// TwinCAT 3 PLC project Plc
// ProgramVersion: 3.1.4026.21
// libraries:
//   [IIN_Base], * (IIN Solutions Oy)
//   Meca500 Functions, * (Iin Solutions Oy)
//   Tc2_DataExchange, * (Beckhoff Automation GmbH)
//   Tc2_MC2, * (Beckhoff Automation GmbH)
//   Tc2_Standard, * (Beckhoff Automation GmbH)
//   Tc2_System, * (Beckhoff Automation GmbH)
//   Tc2_Utilities, * (Beckhoff Automation GmbH)
//   Tc3_EventLogger, * (Beckhoff Automation GmbH)
//   Tc3_Vision, * (Beckhoff Automation GmbH)
// project tree:
//   DUTs/Com/ ST_MecaHmi.TcDUT, ST_ModuleHmi.TcDUT, ST_Module_PlcCom.TcDUT, ST_Module_PlcComIn.TcDUT, ST_Module_PlcComOut.TcDUT, ST_StationHmi.TcDUT
//   DUTs/ E_MecaStatus.TcDUT, ST_Recipes.TcDUT, ST_Recipe_AssemblyData.TcDUT
//   GVLs/ Color.TcGVL, Err.TcGVL, Trig.TcGVL
//   / PlcTask.TcTTO, PlcTaskVis.TcTTO
//   POUs/ FB_ASMT60Functions.TcPOU, FB_GlueState.TcPOU, MAIN.TcPOU
//   POUs/HP/CURING_STATION/ E_CURING_STATION_SEQUENCE_STEPS.TcDUT, E_CURING_STATION_OPERATION_STATE.TcDUT, FB_CuringStation.TcPOU, ST_CURING_STATION_HMI.TcDUT, ST_CURING_STATION_SERVICE.TcDUT, ST_CURING_STATION_STATE.TcDUT, ST_CURING_STATION_SETTINGS.TcDUT
//   POUs/HP/CURING_STATION/HEATER/ E_CURING_STATION_HEATER_CONTROL_STEPS.TcDUT (not stored), FB_CuringStationHeaterControl.TcPOU, ST_CURING_STATION_HEATER_CONTROL_HMI.TcDUT, ST_CURING_STATION_HEATER_CONTROL_SERVICE.TcDUT, ST_CURING_STATION_HEATER_CONTROL_STATE.TcDUT, ST_CURING_STATION_HEATER_CONTROL_STATIC_SETTINGS.TcDUT
//   POUs/HP/CURING_STATION/VISION/Coupler/ E_COUPLER_PROCESSOR_STEPS.TcDUT, FB_CouplerImageProcessor.TcPOU, I_ImageProcessor.TcIO, ST_COUPLER_DETECT_SETTINGS.TcDUT
//   POUs/HP/CURING_STATION/VISION/ E_GIGE_CAM_HANDLER_SEQ_STEPS.TcDUT, E_NORMAL_CAM_HANDLER_SEQ_STEPS.TcDUT, FB_GigECamHandler.TcPOU, FB_CuringStationCameraHandler.TcPOU, ST_LASER_TEST_SETTINGS.TcDUT, ST_NORMAL_CAM_HANDLER_HMI.TcDUT, ST_NORMAL_CAM_HANDLER_SERVICE.TcDUT, ST_NORMAL_CAM_HANDLER_SETTINGS.TcDUT, ST_TEST_SETTING.TcDUT, ST_UNDERLIGHT_TEST_SETTINGS.TcDUT, VISION_PARAMS.TcGVL
//   POUs/HP/CURING_STATION/VISION/GenericCameraHandler/ E_GENERIC_CAM_HANDLER_SEQ_STEPS.TcDUT, FB_GenericCameraHandler.TcPOU
//   POUs/HP/CURING_STATION/VISION/HelperFunctions/ FC_CalculateCenterPoint.TcPOU, FC_CalculateYCenterPoint.TcPOU (not stored), FC_ExtractFromContainerAndCalculateAvg.TcPOU
//   POUs/HP/CURING_STATION/VISION/Mirror/ E_MIRROR_PROCESSOR_STEPS.TcDUT, FB_MirrorImageProcessor.TcPOU, FC_GetCameraScalingFactor.TcPOU, I_MirrorImageProcessor.TcIO, ST_MIRROR_DETECT_SETTINGS.TcDUT
//   POUs/HP/GVL/ HEATER_CONTROL_SETTINGS.TcGVL, HMI.TcGVL, MAIN_VISION_COMM_VARS.TcGVL
//   POUs/HP/ P_Heaters.TcPOU
//   POUs/Meca500/ FB_linearAxisFunctions.TcPOU, FB_MecaStateMachine.TcPOU
//   POUs/Meca500/Op/ E_CurrentState.TcDUT, E_OperatingState.TcDUT, FB_GluingTipPositioning.TcPOU, FB_ManualControl.TcPOU, FB_MecaConf.TcPOU, FB_Operating.TcPOU
//   POUs/Meca500/Op/PoseData/ ST_GluetipCoordinates.TcDUT, ST_GluingPoses.TcDUT, ST_Sts_PoseData.TcDUT, ST_Sts1_PoseData.TcDUT, ST_Sts10_PoseData.TcDUT, ST_Sts2_PoseData.TcDUT, ST_Sts3_PoseData.TcDUT, ST_Sts4_PoseData.TcDUT, ST_Sts5_PoseData.TcDUT, ST_Sts6_PoseData.TcDUT, ST_Sts7_PoseData.TcDUT, ST_Sts8_PoseData.TcDUT, ST_Sts9_PoseData.TcDUT
//   POUs/Meca500/Op/PoseData/Type/ AL82027.TcDUT, AL86068.TcDUT, AL200663.TcDUT, AL200665.TcDUT, AL200664.TcDUT, AL200662.TcDUT
//   POUs/Sts/Com/ FB_DataExchangeRead.TcPOU, FB_RecipeDataExchange.TcPOU, ST_Stations.TcDUT, ST_Sts_PlcCom.TcDUT, ST_Sts_PlcComIn.TcDUT, ST_Sts_PlcComOut.TcDUT
//   POUs/Sts/Datalog/ FB_Datalogger2.TcPOU, FB_Datalogger3.TcPOU, FB_EventLogger.TcPOU, ST_LogEntry.TcDUT
//   POUs/Sts/DUT/ E_MovementState.TcDUT, E_StepperState.TcDUT, E_StsActState.TcDUT, ST_AngleData.TcDUT, ST_Sts_DetectionData.TcDUT, ST_Vis_Laser.TcDUT, ST_Vis_Mirror.TcDUT
//   POUs/Sts/ FB_HeaterControl.TcPOU, FB_Stepper.TcPOU, FB_StsAct.TcPOU
//   POUs/Sts/Vis/ FB_PosImgSts.TcPOU
//   POUs/VisMain/ FB_MidStaion.TcPOU, FB_InfeedCam.TcPOU, FB_OutfeedCam.TcPOU, FB_RejectCam.TcPOU, MAIN_VISION.TcPOU, ST_CouplerImagingData.TcDUT, ST_PalletImagingData.TcDUT

CONFIGURATION Plc
    RESOURCE PLC ON TwinCAT3
        TASK PlcTask(INTERVAL := T#10ms, PRIORITY := 20);
        TASK PlcTaskVis(INTERVAL := T#150ms, PRIORITY := 1);
        PROGRAM MAIN WITH PlcTask : MAIN;
        PROGRAM MAIN_VISION WITH PlcTaskVis : MAIN_VISION;
    END_RESOURCE
END_CONFIGURATION

// ---- DUTs/Com/ST_MecaHmi.TcDUT
TYPE ST_MecaHmi :
STRUCT
	
	bJogToPose			: BOOL;
	aPoseDirect			: ARRAY [1..6] OF REAL;
	bHomeAxis			: BOOL;
	bSetGripperWidth	: BOOL;
	rGripperWidth		: REAL;

// Direct control buttons to robot
	bActivate			: BOOL;
	bDeactivate			: BOOL;
	bErrorReset			: BOOL;
	bManualJog			: BOOL;
	bClearMove			: BOOL;
	bPauseMotion		: BOOL;
	bResumeMotion		: BOOL;
	bDisableEtherCat	: BOOL;
	bToggleGripper		: BOOL;
	bRecoveryMode		: BOOL;

	bJogXPositive		: BOOL;
	bJogXNegative		: BOOL;
	bJogYPositive		: BOOL;
	bJogYNegative		: BOOL;
	bJogZPositive		: BOOL;
	bJogZNegative		: BOOL;
	bJogRxPositive		: BOOL;
	bJogRxNegative		: BOOL;
	bJogRyPositive		: BOOL;
	bJogRyNegative		: BOOL;
	bJogRzPositive		: BOOL;
	bJogRzNegative		: BOOL;
	rJogSpeed			: REAL := 10;
	aCurrentPose		: ARRAY [1..6] OF REAL;
	bJogLinearPositive	: BOOL;
	bJogLinearNegative	: BOOL;
	bLinearJogScreenActive	: BOOL;
	bManualAbsMove : BOOL;
	rManualTargetPos	: REAL;
	
END_STRUCT
END_TYPE

// ---- DUTs/Com/ST_ModuleHmi.TcDUT
TYPE ST_ModuleHmi :
STRUCT
	
	MecaHmi 					: ST_MecaHmi;
	Stations					: ST_StationHmi;
	bModuleProductionStart		: BOOL; // Is always active if assemblies are active
	bModulePlayPause 			: BOOL; // Only used for glue remove
	bProductionStart1To5 		: BOOL; // 
	bProductionStart6To10		: BOOL;
	bProductionStageCompleted	: BOOL; // To indicate that assemblies of 1 to 5 or 6 to 10 are set and more assemblies can be inserted
	bModuleProductionStop		: BOOL;
	bModuleStartup				: BOOL;
	bModuleStartupDone			: BOOL;
	bModuleFault				: BOOL;
	bResetCommunication			: BOOL;
	bResetModuleFault			: BOOL;
	bPowerOff					: BOOL;
	bClearAlarms				: BOOL;
	sOperatingStatus			: STRING;
	bProductionStartFailure		: BOOL;
	bOpenAllLocks				: BOOL;
	bAcOk						: BOOL;
	
	bGlueDispensing				: BOOL;
	bToggleDispensingPressure	: BOOL;
	bDispensingPressed			: BOOL;
	bStartDetection				: BOOL;
	bAllowManDispensing			: BOOL;
	bDetectionSucceeded			: BOOL;
	sTimeSinceDispensing		: STRING;
	bDispensingStageDone		: BOOL;
	
END_STRUCT
END_TYPE

// ---- DUTs/Com/ST_Module_PlcCom.TcDUT
TYPE ST_Module_PlcCom :
STRUCT
	
	stPlcComIn		AT %I*: ST_Module_PlcComIn;
	stPlcComOut		AT %Q*: ST_Module_PlcComOut;

END_STRUCT
END_TYPE

// ---- DUTs/Com/ST_Module_PlcComIn.TcDUT
TYPE ST_Module_PlcComIn :
STRUCT
	bEstopOk	: BOOL;
	bSafetyOk  : BOOL;
	bUpsStatusOk	: BOOL;	
	bLinearAxisHomingSensor : BOOL;
	bRobotGripperSensor : BOOL;
	bRobotPower	: BOOL;
	
	bGlueDoorUpperLockOpen		: BOOL;
	bGlueDoorUpperLockClosed	: BOOL;
	bGlueDoorLowerLockOpen		: BOOL;
	bGlueDoorLowerLockClosed	: BOOL;
	
	bMainDoorLockOpen			: BOOL;
	bMainDoorLockClosed			: BOOL;
	bPassLockOpen				: BOOL;
	bPassLockClosed				: BOOL;
	bInfeedLockOpen				: BOOL;
	bInfeedLockClosed			: BOOL;
	bRejectLockOpen				: BOOL;
	bRejectLockClosed			: BOOL;
	
	bUpsAlarm					: BOOL;
	bAcOk						: BOOL;
	iModuleTemp					: INT;
	bGlueStopHome				: BOOL;
END_STRUCT
END_TYPE

// ---- DUTs/Com/ST_Module_PlcComOut.TcDUT
TYPE ST_Module_PlcComOut :
STRUCT
	bTriggerGluing1			: BOOL;
	bLaserPointers1To5		: BOOL;
	bLaserPointers5To10		: BOOL;
	bResetButtonLight		: BOOL;
	bMecaReset				: BOOL;
	bRobotSwStop			: BOOL;
	
	bRingLightGlue			: BOOL;
	bRingLightInfeed		: BOOL;
	bRingLightPass			: BOOL;
	bRingLightReject		: BOOL;
	
	bGlueDoorLock			: BOOL;
	bHatchesLock			: BOOL;
	bPowerOff				: BOOL;
	bGlueStopValve			: BOOL;
	bGlueSelectingValve		: BOOL;
END_STRUCT
END_TYPE

// ---- DUTs/Com/ST_StationHmi.TcDUT
TYPE ST_StationHmi :
STRUCT
		
	bActivateStation1 : BOOL := TRUE;
	bActivateStation2 : BOOL := TRUE;
	bActivateStation3 : BOOL := TRUE;
	bActivateStation4 : BOOL := TRUE;
	bActivateStation5 : BOOL := TRUE;
	bActivateStation6 : BOOL := TRUE;
	bActivateStation7 : BOOL := TRUE;
	bActivateStation8 : BOOL := TRUE;
	bActivateStation9 : BOOL := TRUE;
	bActivateStation10 : BOOL := TRUE;
	
	tAssemmblyTime1				: STRING;
	tAssemmblyTime2				: STRING;
	tAssemmblyTime3				: STRING;
	tAssemmblyTime4				: STRING;
	tAssemmblyTime5				: STRING;
	tAssemmblyTime6				: STRING;
	tAssemmblyTime7				: STRING;
	tAssemmblyTime8				: STRING;
	tAssemmblyTime9				: STRING;
	tAssemmblyTime10			: STRING;
	
	bReleaseHolders1			: BOOL;
	bReleaseHolders2			: BOOL;
	bReleaseHolders3			: BOOL;
	bReleaseHolders4			: BOOL;
	bReleaseHolders5			: BOOL;
	bReleaseHolders6			: BOOL;
	bReleaseHolders7			: BOOL;
	bReleaseHolders8			: BOOL;
	bReleaseHolders9			: BOOL;
	bReleaseHolders10			: BOOL;
	
END_STRUCT
END_TYPE

// ---- DUTs/E_MecaStatus.TcDUT
{attribute 'qualified_only'}
{attribute 'strict'}
{attribute 'to_string'}
TYPE E_MecaStatus :
(
	Offline,
	Conf,
	Idle,
	Operating,
	Home,
	HmiManual,
	GluingpPos
);
END_TYPE

// ---- DUTs/ST_Recipes.TcDUT
TYPE ST_Recipes :
STRUCT
	Station1To5		: ST_Recipe_AssemblyData;
	Station5To10	: ST_Recipe_AssemblyData;
END_STRUCT
END_TYPE

// ---- DUTs/ST_Recipe_AssemblyData.TcDUT
TYPE ST_Recipe_AssemblyData :
STRUCT
	rGalvoThickness			: REAL;
	rMirrorDimensions : ARRAY [0..3] OF REAL; //[0] Width at mirror girp center position (gripperWidth), [1] Width, [2] height, [3] Thickness
 	
	// To enable new mirror variations to be added only based on offset values
	rMirrorGripPointOffsetToEdgeX	: REAL; // Distance from grip centerpoint to mirror edge on the direction of the gluing side
	rMirrorCenterOffsetToWeightCenterY : REAL; // Distance from mirror weight centerpoint to mirror width centerpoint.
	rLaserPointSetValue	: REAL;
	rCouplerGroveDepth	: REAL; // Depth from CAD files of the couplers
	// Coupler detection variables
	rThreshold			: LREAL;
	aStartPointCoupler					: TcVnPoint2_REAL;
	aEndPointCoupler					: TcVnPoint2_REAL;
	rSearchLineDist							: REAL;
	//
	wPalletBinary		: WORD;
	sAssemblyType	: STRING;
	sMotorType	: STRING;
	sMirrorType	: STRING;
	sGlueType	: STRING;
	sCouplerType : STRING;
	
	// for data exchange
	bTrigCam1	: BOOL;
	bTrigCam2	: BOOL;
	bTrigCam3	: BOOL;
	bTrigCam4	: BOOL;
	bTrigCam5	: BOOL;
	bTrigCam6	: BOOL;
	bTrigCam7	: BOOL;
	bTrigCam8	: BOOL;
	bTrigCam9	: BOOL;
	bTrigCam10	: BOOL;
	
END_STRUCT
END_TYPE

// ---- POUs/HP/CURING_STATION/E_CURING_STATION_SEQUENCE_STEPS.TcDUT
{attribute 'qualified_only'}
{attribute 'strict'}
{attribute 'to_string'}
TYPE E_CURING_STATION_SEQUENCE_STEPS :
(
	INIT := 0,
	
	STARTUP_TEST_DO_ECCENTRIC_WHEEL_HOMING,
	
	STARTUP_TEST_TEST_SLIDER_TO_WORK,
	STARTUP_TEST_TEST_SLIDER_TO_HOME,
	
	STARTUP_TEST_TEST_GRIPPER_TO_WORK,
	STARTUP_TEST_TEST_GRIPPER_TO_HOME,
	
	STARTUP_TEST_TEST_UNDERLIGHT,
	
	STARTUP_TEST_TEST_LASER,
	
	STARTUP_TEST_TEST_HEATER,

	STARTUP_TEST_DONE,

	STARTUP_TEST_FAIL,	
	
	OPERATIONAL
	
);
END_TYPE

// ---- POUs/HP/CURING_STATION/E_CURING_STATION_OPERATION_STATE.TcDUT
{attribute 'qualified_only'}
{attribute 'strict'}
{attribute 'to_string'}
TYPE E_CURING_STATION_OPERATION_STATE :
(
	INACTIVE := 0,
	
	OPERATIONAL,
	
	FAULTED
);
END_TYPE

// ---- POUs/HP/CURING_STATION/HEATER/ST_CURING_STATION_HEATER_CONTROL_HMI.TcDUT
TYPE ST_CURING_STATION_HEATER_CONTROL_HMI :
STRUCT
	state:				ST_CURING_STATION_HEATER_CONTROL_STATE;
	service:			ST_CURING_STATION_HEATER_CONTROL_SERVICE;
	
	ai:						ST_AI_HMI;
//	regularThermostat:		ST_THERMOSTAT_HMI;
	specialThermostat:		ST_TIME_PROPORTIONAL_THERMOSTAT_HMI;
END_STRUCT
END_TYPE

// ---- POUs/HP/CURING_STATION/HEATER/ST_CURING_STATION_HEATER_CONTROL_SERVICE.TcDUT
TYPE ST_CURING_STATION_HEATER_CONTROL_SERVICE :
STRUCT
	
END_STRUCT
END_TYPE

// ---- POUs/HP/CURING_STATION/HEATER/ST_CURING_STATION_HEATER_CONTROL_STATE.TcDUT
TYPE ST_CURING_STATION_HEATER_CONTROL_STATE :
STRUCT
	enabled:					BOOL;
	heat:						BOOL;
	fan:						BOOL;
	tempInC:					REAL;
//		tempInF:					REAL;
	testTemperatureReached:		BOOL; 
	workTemperatureReached:		BOOL;
	stationId:					UDINT; 
END_STRUCT
END_TYPE

// ---- POUs/HP/CURING_STATION/HEATER/ST_CURING_STATION_HEATER_CONTROL_STATIC_SETTINGS.TcDUT
TYPE ST_CURING_STATION_HEATER_CONTROL_STATIC_SETTINGS :
STRUCT
	testTemperature:			REAL := 28.0;
	workTemperature:			REAL := 50.0;
	hysteresis:					REAL := 2.0;	// If temp within this value, temp is 'reached'
	
	pFactor:					REAL := 3;		// Temp diff * pFactor = power output (just like a PID controller but without the ID)
	minPowerProcent:			REAL := 20;		// If this were a PID controller, we need 20% to keep the constant heat (at target setpoint)
	maxPowerProcent:			REAL := 80;		// To limit the output (in case the heating element is too powerfull)

	cycleTime:					TIME := T#20S;	// 100% control = HEAT is on for this amount of cycle time, 50% results in 10sec ON and 10s OFF
	nrOfStations:				UDINT := 10;	// Used to calculate a start delay for the heaters to go on -> so FUSE won't blow
END_STRUCT
END_TYPE

// ---- POUs/HP/CURING_STATION/ST_CURING_STATION_HMI.TcDUT
TYPE ST_CURING_STATION_HMI :
STRUCT
	state:			ST_CURING_STATION_STATE;
	service:		ST_CURING_STATION_SERVICE;
	settings:		ST_CURING_STATION_SETTINGS;
	
	cyls:			ARRAY[0..1] OF ST_CYL_HMI;
	heater:			ST_CURING_STATION_HEATER_CONTROL_HMI;
END_STRUCT
END_TYPE

// ---- POUs/HP/CURING_STATION/ST_CURING_STATION_SERVICE.TcDUT
TYPE ST_CURING_STATION_SERVICE :
STRUCT
	enable:	BOOL;		// Setting on/off will enable the station
END_STRUCT
END_TYPE

// ---- POUs/HP/CURING_STATION/ST_CURING_STATION_STATE.TcDUT
TYPE ST_CURING_STATION_STATE :
STRUCT
	stationId:				UDINT; 
	operationState:			E_CURING_STATION_OPERATION_STATE;
END_STRUCT
END_TYPE

// ---- POUs/HP/CURING_STATION/ST_CURING_STATION_SETTINGS.TcDUT
TYPE ST_CURING_STATION_SETTINGS :
STRUCT
END_STRUCT
END_TYPE

// ---- POUs/HP/CURING_STATION/VISION/Coupler/E_COUPLER_PROCESSOR_STEPS.TcDUT
{attribute 'qualified_only'}
{attribute 'strict'}
{attribute 'to_string'}
TYPE E_COUPLER_PROCESSOR_STEPS :
(
	INIT := 0,
	
	LOCATE_EDGE1,
	
	LOCATE_EDGE2,

	LOCATE_EDGE3,
	
	DRAW_POINTS,
	
	MAKE_DISPLAYABLE,
	
	DONE,
	
	ERROR,
	
	END
	
);
END_TYPE

// ---- POUs/HP/CURING_STATION/VISION/Coupler/ST_COUPLER_DETECT_SETTINGS.TcDUT
TYPE ST_COUPLER_DETECT_SETTINGS :
STRUCT
//	startPoint:		TcVnPoint2_REAL := [1000, 550];
//	endPoint:		TcVnPoint2_REAL := [550, 1000];
	
//	minStrength:	REAL := 45;
//	searchLines:	UDINT := 5;
END_STRUCT
END_TYPE

// ---- POUs/HP/CURING_STATION/VISION/E_GIGE_CAM_HANDLER_SEQ_STEPS.TcDUT
{attribute 'qualified_only'}
{attribute 'strict'}
{attribute 'to_string'}
TYPE E_GIGE_CAM_HANDLER_SEQ_STEPS :
(
	INIT,
	
	RESET_CAMERA,
	
	READY_FOR_OPERATION,
	
	TRIGGER_CAMERA,
	
	START_ACQUISITION,
	
	ACQUIRING,
	
	DO_COLOR_CONVERSION,
	
	ACQUIRED,
	
	ERROR,
	
	DONE,
	
	END
);
END_TYPE

// ---- POUs/HP/CURING_STATION/VISION/E_NORMAL_CAM_HANDLER_SEQ_STEPS.TcDUT
{attribute 'qualified_only'}
{attribute 'strict'}
{attribute 'to_string'}
TYPE E_NORMAL_CAM_HANDLER_SEQ_STEPS :
(
	INIT := 0,

	UNDER_LIGHT_TEST_ENABLE_LIGHT,
	UNDER_LIGHT_TEST_IMAGE_ACQUIRE,
	UNDER_LIGHT_TEST_IMAGE_PROCESSING,
	UNDER_LIGHT_TEST_OK,
	UNDER_LIGHT_TEST_FAILED,

	LASER_LIGHT_TEST_ENABLE_LIGHT,
	LASER_LIGHT_TEST_IMAGE_ACQUIRE,
	LASER_LIGHT_TEST_IMAGE_PROCESSING,
	LASER_LIGHT_TEST_OK,
	LASER_LIGHT_TEST_FAILED,
	
	COUPLER_DETECT_ENABLE_LIGHT,
	COUPLER_DETECT_IMAGE_ACQUIRE,
	COUPLER_DETECT_IMAGE_PROCESSING,
	COUPLER_DETECT_DONE,
	COUPLER_DETECT_FAILED,

	MIRROR_DETECT_ENABLE_LIGHT,
	MIRROR_DETECT_IMAGE_ACQUIRE,
	MIRROR_DETECT_IMAGE_PROCESSING,
	MIRROR_DETECT_DONE,
	MIRROR_DETECT_FAILED,
	
	
	END
);
END_TYPE

// ---- POUs/HP/CURING_STATION/VISION/GenericCameraHandler/E_GENERIC_CAM_HANDLER_SEQ_STEPS.TcDUT
{attribute 'qualified_only'}
{attribute 'strict'}
{attribute 'to_string'}
TYPE E_GENERIC_CAM_HANDLER_SEQ_STEPS :
(
	INIT := 0,

	UNDER_LIGHT_TEST_ENABLE_LIGHT,
	UNDER_LIGHT_TEST_IMAGE_ACQUIRE,
	UNDER_LIGHT_TEST_IMAGE_PROCESSING,
	UNDER_LIGHT_TEST_OK,
	UNDER_LIGHT_TEST_FAILED,

	LASER_LIGHT_TEST_ENABLE_LIGHT,
	LASER_LIGHT_TEST_IMAGE_ACQUIRE,
	LASER_LIGHT_TEST_IMAGE_PROCESSING,
	LASER_LIGHT_TEST_OK,
	LASER_LIGHT_TEST_FAILED,
	
	COUPLER_DETECT_ENABLE_LIGHT,
	COUPLER_DETECT_IMAGE_ACQUIRE,
	COUPLER_DETECT_IMAGE_PROCESSING,
	COUPLER_DETECT_DONE,
	COUPLER_DETECT_FAILED,

	MIRROR_DETECT_ENABLE_LIGHT,
	MIRROR_DETECT_IMAGE_ACQUIRE,
	MIRROR_DETECT_IMAGE_PROCESSING,
	MIRROR_DETECT_DONE,
	MIRROR_DETECT_FAILED,
	
	
	END
);
END_TYPE

// ---- POUs/HP/CURING_STATION/VISION/Mirror/E_MIRROR_PROCESSOR_STEPS.TcDUT
{attribute 'qualified_only'}
{attribute 'strict'}
{attribute 'to_string'}
TYPE E_MIRROR_PROCESSOR_STEPS :
(
	INIT := 0,
	
	CALC_CENTER_POINT_OFFSET,
	
	FIND_UPPER_EDGE,
	
	FIND_LOWER_EDGE,

	DRAW_POINTS,
	
	MAKE_DISPLAYABLE,
	
	DONE,
	
	ERROR,
	
	END
	
);
END_TYPE

// ---- POUs/HP/CURING_STATION/VISION/Mirror/ST_MIRROR_DETECT_SETTINGS.TcDUT
TYPE ST_MIRROR_DETECT_SETTINGS :
STRUCT
//	startPoint:		TcVnPoint2_REAL := [1000, 550];
//	endPoint:		TcVnPoint2_REAL := [550, 1000];
	
//	minStrength:	REAL := 45;
//	searchLines:	UDINT := 5;
END_STRUCT
END_TYPE

// ---- POUs/HP/CURING_STATION/VISION/ST_LASER_TEST_SETTINGS.TcDUT
TYPE ST_LASER_TEST_SETTINGS :
STRUCT
	height:		UDINT := 20;
	width:		UDINT := 20;
	x:			UDINT := 800;
	y:			UDINT := 900;
	
	threshold:	LREAL := 230;		// Average pixel value for the test to be successfull
END_STRUCT
END_TYPE

// ---- POUs/HP/CURING_STATION/VISION/ST_NORMAL_CAM_HANDLER_HMI.TcDUT
TYPE ST_NORMAL_CAM_HANDLER_HMI :
STRUCT
END_STRUCT
END_TYPE

// ---- POUs/HP/CURING_STATION/VISION/ST_NORMAL_CAM_HANDLER_SERVICE.TcDUT
TYPE ST_NORMAL_CAM_HANDLER_SERVICE :
STRUCT
	doUnderLightTest:		BOOL;
	doLaserTest:			BOOL;
END_STRUCT
END_TYPE

// ---- POUs/HP/CURING_STATION/VISION/ST_NORMAL_CAM_HANDLER_SETTINGS.TcDUT
TYPE ST_NORMAL_CAM_HANDLER_SETTINGS :
STRUCT
	underLightTest:	ST_UNDERLIGHT_TEST_SETTINGS;
	laserTest:		ST_LASER_TEST_SETTINGS;
END_STRUCT
END_TYPE

// ---- POUs/HP/CURING_STATION/VISION/ST_TEST_SETTING.TcDUT
TYPE ST_TEST_SETTING :
STRUCT
	height:		UDINT;
	width:		UDINT;
	x:			UDINT;
	y:			UDINT;
END_STRUCT
END_TYPE

// ---- POUs/HP/CURING_STATION/VISION/ST_UNDERLIGHT_TEST_SETTINGS.TcDUT
TYPE ST_UNDERLIGHT_TEST_SETTINGS :
STRUCT
	height:		UDINT := 200;
	width:		UDINT := 200;
	x:			UDINT := 1800;
	y:			UDINT := 900;
	
	threshold:	LREAL := 230;		// Average pixel value for the test to be successfull
END_STRUCT
END_TYPE

// ---- POUs/Meca500/Op/E_CurrentState.TcDUT
{attribute 'qualified_only'}
{attribute 'strict'}
{attribute 'to_string'}
TYPE E_CurrentState :
(
	Init,
	GalvoHandling,
	MirrorAdj,
	FinishedProduct

);
END_TYPE

// ---- POUs/Meca500/Op/E_OperatingState.TcDUT
{attribute 'qualified_only'}
{attribute 'strict'}
{attribute 'to_string'}
TYPE E_OperatingState :
(
	Init,
	MoveLinAxis,
	SetPoses,
	OperatingGalvo14mm,
	OperatingGalvo10mm,
	MirrorAdjustment,
	FinishedHandling14mm,
	FinishedHandling10mm
);
END_TYPE

// ---- POUs/Meca500/Op/PoseData/ST_GluetipCoordinates.TcDUT
TYPE ST_GluetipCoordinates :
STRUCT
	X : REAL;
	Y : REAL;
	Z : REAL;
END_STRUCT
END_TYPE

// ---- POUs/Meca500/Op/PoseData/ST_GluingPoses.TcDUT
TYPE ST_GluingPoses :
STRUCT
	AL200662: AL200662;
	AL82027: AL82027;
END_STRUCT
END_TYPE

// ---- POUs/Meca500/Op/PoseData/ST_Sts_PoseData.TcDUT
TYPE ST_Sts_PoseData :
STRUCT
	// Pickup positions and pass pallet positions are all station related. So from pallet position 1 it is only possible to place it to curing station 1 and to pass pallet position 1.
	// Positions are claculated with 'Machine cordinate chart' Excel
	
	aPoseSmallMotorPickupSt1 : ARRAY [1..6] OF REAL := [-144.652, 129 , 110.5 , 0, -90 ,0] ; // Pose before gripper in to the pallet picking position
	aPoseSmallMotorPickupSt2 : ARRAY [1..6] OF REAL := [-144.652, 129 , 110.5 , 0, -90 ,0] ; // Pose before gripper grip, or pose after gripper grip
	aPoseSmallMotorPickupSt3 : ARRAY [1..6] OF REAL := [-144.652, 129 , 110.5 , 0, -90 ,0] ; // Pose gripper grip
	
	aPoseSmallMotorPlaceSt1 : ARRAY [1..6] OF REAL; // Pose before Small motor in station
	aPoseSmallMotorPlaceSt2 : ARRAY [1..6] OF REAL; // Pose Small motor in station
	rLinPosPlace : LREAL; // Linear axis position for placing functions for selected station

	aPoseMirrorAdj : ARRAY[1..6] OF REAL; // Pose where final position of left mirror is saved in case position adjustment is needed.
	
	aPoseLargeMotorPickupSt1	: ARRAY [1..6] OF REAL := [-95,-150.45 , 110.5 , 0, -90 ,0]; // POSE BEFORE ACTUAL GRIP POSITION -108.2
	aPoseLargeMotorPickupSt2	: ARRAY [1..6] OF REAL := [-128.2,-150.45 , 110.5 , 0, -90 ,0];// ACTUAL GRIP POSITION
	aPoseLargeMotorPickupSt3	: ARRAY [1..6] OF REAL := [-128.2,-150.45 , 200.5 , 0, -90 ,0];// MOTOR LIFT FROM PALLET
	rLinPosMotorPickup				: LREAL := 120; // Linear axis position for pickup functions for selected station
	
	aPoseLargeMotorPlaceSt1	: ARRAY [1..6] OF REAL := [-144.652, 129 ,165.6645  , -180 , 0 , 90]; // POSE BEFORE ACTULA LEAVING POSITION
	aPoseLargeMotorPlaceSt2	: ARRAY [1..6] OF REAL := [-73.8605, 140 ,165.6645  , -180 , 0 , 90]; // ACTUAL POSITION FOR LEAVING MOTOR AT CURING STATION
	aPoseLargeMotorPlaceSt3	: ARRAY [1..6] OF REAL := [-73.8605, 140 ,200  , -180 , 0 , 90]; // POSE AFTER LEAVING MOTOR AT CURING STATION
	
	aPoseMirrorPickupSt1	: ARRAY [1..6] OF REAL := [-159.1,-91.5 , 200 ,180, 0 ,0]; // POSE BEFORE ACTUAL GRIP POSITION
	aPoseMirrorPickupSt2	: ARRAY [1..6] OF REAL := [-159.1,-91.5 , 186.9757 ,180, 0 ,0];// ACTUAL GRIP POSITION 187.1757
	rLinPosMirrorPickup				: LREAL := 120; // Linear axis position for pickup functions for selected station
	
	aPoseMirrorPlaceSt1	: ARRAY [1..6] OF REAL := [-72, 192.8 ,200.3  , -180 , 0 , 90]; // POSE BEFORE INSERTIN MIRROR IN STATION
	aPoseMirrorPlaceSt2	: ARRAY [1..6] OF REAL := [-72, 192.8 ,173.55  , -180 , 0 , 90]; // POSE MIRROR IN STATION BUT NOT INSERTED TO MOTOR  192.8, 173.45
	aPoseMirrorPlaceSt3	: ARRAY [1..6] OF REAL := [-72, 189.4545 ,173.95  , -180 , 0 , 90]; // POSE MIRROR INSERTED TO MOTOR
 	
// 	aPoseSmallMirrorPlaceSt1	: ARRAY [1..6] OF REAL := [-72, 192.8 ,200.3  , -180 , 0 , 90]; // POSE BEFORE INSERTIN MIRROR IN STATION
// 	aPoseSmallMirrorPlaceSt2	: ARRAY [1..6] OF REAL := [-72, 192.8 ,173.55  , -180 , 0 , 90]; // POSE MIRROR IN STATION BUT NOT INSERTED TO MOTOR  192.8, 173.45
// 	aPoseSmallMirrorPlaceSt3	: ARRAY [1..6] OF REAL := [-72, 189.4545 ,173.95  , -180 , 0 , 90]; // POSE MIRROR INSERTED TO MOTOR
	
	aPosePassedLargeSt1 		: ARRAY [1..6] OF REAL := [-72.2, 189.4545 ,173.95  , -180 , 0 , 90];
	aPosePassedLargeSt2			: ARRAY [1..6] OF REAL := [-72.2, 189.4545 ,173.95  , -180 , 0 , 90];
	aPosePassedLargeSt3			: ARRAY [1..6] OF REAL := [-72.2, 189.4545 ,173.95  , -180 , 0 , 90];
	
	aPosePassedSmallSt1			: ARRAY [1..6] OF REAL := [-72.2, 189.4545 ,173.95  , -180 , 0 , 90];
	aPosePassedSmallSt2			: ARRAY [1..6] OF REAL := [-72.2, 189.4545 ,173.95  , -180 , 0 , 90];
	aPosePassedSmallSt3			: ARRAY [1..6] OF REAL := [-72.2, 189.4545 ,173.95  , -180 , 0 , 90];
	aPosePassedSmallSt4			: ARRAY [1..6] OF REAL := [-72.2, 189.4545 ,173.95  , -180 , 0 , 90];
	
	rLinPosPalletPass : LREAL; // Linear axis position for placing passed assembly for selected station
	rLinPosPalletReject : LREAL; // Linear axis position for placing rejected assembly for selected station
	
END_STRUCT
END_TYPE

// ---- POUs/Meca500/Op/PoseData/ST_Sts1_PoseData.TcDUT
TYPE ST_Sts1_PoseData :
STRUCT
	
	aPoseSmallMotorPickupSt1 : ARRAY [1..6] OF REAL := [-220.552, 67.9 , 150, 180, -20 ,0] ; // Pose before gripper in to the pallet picking position
	aPoseSmallMotorPickupSt2 : ARRAY [1..6] OF REAL := [-220.552, 67.9 , 111.4134, 180, -20 ,0] ;  // Pose before gripper grip, or pose after gripper grip
	aPoseSmallMotorPickupSt3 : ARRAY [1..6] OF REAL := [-222.713, 67.9 , 112.2, 180, -20 ,0] ; //  Pose gripper grip CAN NOT BE MOVEPOSE
	rLinPosSmallMotorPickup				: LREAL := 80; // Linear axis position for pickup functions for selected station
	
	aPoseSmallMotorPlaceSt1 : ARRAY [1..6] OF REAL := [-73.2, 168.6 ,110.6 , 180, 0 ,90] ; // Pose before Small motor in station
	aPoseSmallMotorPlaceSt2 : ARRAY [1..6] OF REAL  := [-73.2, 168.6 ,67.6 , 180, 0 ,90]; // Pose Small motor in station
	rLinPosPlace : LREAL := 10; // Linear axis position for placing functions for selected station

	aPoseMirrorAdj : ARRAY[1..6] OF REAL; // Pose where final position of left mirror is saved in case position adjustment is needed.
	
	aPoseLargeMotorPickupSt1	: ARRAY [1..6] OF REAL := [-124.609, 117.800 , 101.6 , 0, -90 ,0]; // POSE BEFORE ACTUAL GRIP POSITION -108.2
	aPoseLargeMotorPickupSt2	: ARRAY [1..6] OF REAL := [-224.609, 117.800 , 101.6 , 0, -90 ,0];// ACTUAL GRIP POSITION
	aPoseLargeMotorPickupSt3	: ARRAY [1..6] OF REAL := [-224.609, 117.800 , 201.6 , 0, -90 ,0];// MOTOR LIFT FROM PALLET
	rLinPosMotorPickup				: LREAL := 120; // Linear axis position for pickup functions for selected station
	
	aPoseLargeMotorPlaceSt1	: ARRAY [1..6] OF REAL := [-73.3, 80 , 67.6 , 180, 0 ,90]; // POSE BEFORE ACTULA LEAVING POSITION '
	aPoseLargeMotorPlaceSt2	: ARRAY [1..6] OF REAL := [-73.3, 146 , 67.6 , 180, 0 ,90]; // ACTUAL POSITION FOR LEAVING MOTOR AT CURING STATION '
	aPoseLargeMotorPlaceSt3	: ARRAY [1..6] OF REAL := [-73.3, 146 , 100.6 , 180, 0 ,90]; // POSE AFTER LEAVING MOTOR AT CURING STATION '
	
	aPoseMirrorPickupSt1	: ARRAY [1..6] OF REAL := [-158.84, 76.3 , 120, 181, 0 ,0]; // POSE BEFORE ACTUAL GRIP POSITION
	aPoseMirrorPickupSt2	: ARRAY [1..6] OF REAL := [-158.84, 76.3 , 81.55, 181, 0 ,0];// ACTUAL GRIP POSITION 187.1757
	rLinPosMirrorPickup				: LREAL := 80; // Linear axis position for pickup functions for selected station
	
 	aPoseG10MirrorPlaceSt1	: ARRAY [1..6] OF REAL := [-73.3, 190.6 ,117.4 , 180, 0 ,90]; // POSE BEFORE INSERTIN MIRROR IN STATION'
 	aPoseG10MirrorPlaceSt2	: ARRAY [1..6] OF REAL := [-73.3, 188.2 ,70.4 , -180, 0 ,90]; // POSE MIRROR IN STATION BUT NOT INSERTED TO MOTOR '
 	aPoseg10MirrorPlaceSt3	: ARRAY [1..6] OF REAL := [-73.3, 187 ,68.6 , -179, 0 ,90]; // POSE MIRROR INSERTED TO MOTOR'
	
	aPoseG14MirrorPlaceSt1	: ARRAY [1..6] OF REAL := [-73.3, 190.6 ,117.4 , 180, 0 ,90]; // POSE BEFORE INSERTIN MIRROR IN STATION'
	aPoseG14MirrorPlaceSt2	: ARRAY [1..6] OF REAL := [-73.3, 191.6 ,70.4 , -170, 0 ,90]; // POSE MIRROR IN STATION BUT NOT INSERTED TO MOTOR '
	aPoseg14MirrorPlaceSt3	: ARRAY [1..6] OF REAL := [-73.3, 190.1 ,68.6 , -178.5, -0.2 ,90]; // POSE MIRROR INSERTED TO MOTOR'
	
	aPosePassedLargeSt1 		: ARRAY [1..6] OF REAL := [-213.4, 62.25 , 141.45, 180, -20 ,0]; // In and out of pallet
	aPosePassedLargeSt2			: ARRAY [1..6] OF REAL := [-223.4, 62.25 , 101.45, 180, -20 ,0]; // before leaving position
	aPosePassedLargeSt3			: ARRAY [1..6] OF REAL := [-228, 62.25 ,97.79, 180, -20 ,0]; // Leaving position
	
	aPosePassedSmallSt1			: ARRAY [1..6] OF REAL := [-243.3, 42.14 ,157.0, -180, -20 ,0];
	aPosePassedSmallSt2			: ARRAY [1..6] OF REAL := [-243.3, 42.14 ,127.0, -180, -20 ,0];
	aPosePassedSmallSt3			: ARRAY [1..6] OF REAL := [-250.57, 42.14 ,105.640 , -180, -20 ,0];
	
	rLinPosPalletPass : LREAL := 280; // Linear axis position for placing passed assembly for selected station
	rLinPosPalletReject : LREAL; // Linear axis position for placing rejected assembly for selected station
	
END_STRUCT
END_TYPE

// ---- POUs/Meca500/Op/PoseData/ST_Sts10_PoseData.TcDUT
TYPE ST_Sts10_PoseData :
STRUCT
	
	aPoseSmallMotorPlaceSt1 : ARRAY [1..6] OF REAL; // Pose before Small motor in station
	aPoseSmallMotorPlaceSt2 : ARRAY [1..6] OF REAL; // Pose Small motor in station
	rLinPosPlace : LREAL; // Linear axis position for placing functions for selected station

	aPoseMirrorAdj : ARRAY[1..6] OF REAL; // Pose where final position of left mirror is saved in case position adjustment is needed.
	
	aPoseLargeMotorPickupSt1	: ARRAY [1..6] OF REAL := [-95,-150.45 , 110.5 , 0, -90 ,0]; // POSE BEFORE ACTUAL GRIP POSITION -108.2
	aPoseLargeMotorPickupSt2	: ARRAY [1..6] OF REAL := [-128.2,-150.45 , 110.5 , 0, -90 ,0];// ACTUAL GRIP POSITION
	aPoseLargeMotorPickupSt3	: ARRAY [1..6] OF REAL := [-128.2,-150.45 , 200.5 , 0, -90 ,0];// MOTOR LIFT FROM PALLET
	rLinPosPickup				: LREAL; // Linear axis position for pickup functions for selected station
	
	aPoseLargeMotorPlaceSt1	: ARRAY [1..6] OF REAL := [-73.8605, 110 ,165.6645  , -180 , 0 , 90]; // POSE BEFORE ACTULA LEAVING POSITION
	aPoseLargeMotorPlaceSt2	: ARRAY [1..6] OF REAL := [-73.8605, 140 ,165.6645  , -180 , 0 , 90]; // ACTUAL POSITION FOR LEAVING MOTOR AT CURING STATION
	aPoseLargeMotorPlaceSt3	: ARRAY [1..6] OF REAL := [-73.8605, 140 ,200  , -180 , 0 , 90]; // POSE AFTER LEAVING MOTOR AT CURING STATION
	
	aPoseMirrorPickupSt1	: ARRAY [1..6] OF REAL := [-159.1,-91.5 , 200 ,180, 0 ,0]; // POSE BEFORE ACTUAL GRIP POSITION
	aPoseMirrorPickupSt2	: ARRAY [1..6] OF REAL := [-159.1,-91.5 , 186.9757 ,180, 0 ,0];// ACTUAL GRIP POSITION 187.1757
	
	aPoseMirrorPlaceSt1	: ARRAY [1..6] OF REAL := [-72.2, 192.8 ,200.3  , -180 , 0 , 90]; // POSE BEFORE INSERTIN MIRROR IN STATION
	aPoseMirrorPlaceSt2	: ARRAY [1..6] OF REAL := [-72.2, 192.8 ,173.55  , -180 , 0 , 90]; // POSE MIRROR IN STATION BUT NOT INSERTED TO MOTOR  192.8, 173.45
	aPoseMirrorPlaceSt3	: ARRAY [1..6] OF REAL := [-72.2, 189.4545 ,173.95  , -180 , 0 , 90]; // POSE MIRROR INSERTED TO MOTOR
	
	aPosePassedLargeSt1 		: ARRAY [1..6] OF REAL := [-72.2, 189.4545 ,173.95  , -180 , 0 , 90];
	aPosePassedLargeSt2			: ARRAY [1..6] OF REAL := [-72.2, 189.4545 ,173.95  , -180 , 0 , 90];
	aPosePassedLargeSt3			: ARRAY [1..6] OF REAL := [-72.2, 189.4545 ,173.95  , -180 , 0 , 90];
	
	aPosePassedSmallSt1			: ARRAY [1..6] OF REAL := [-72.2, 189.4545 ,173.95  , -180 , 0 , 90];
	aPosePassedSmallSt2			: ARRAY [1..6] OF REAL := [-72.2, 189.4545 ,173.95  , -180 , 0 , 90];
	aPosePassedSmallSt3			: ARRAY [1..6] OF REAL := [-72.2, 189.4545 ,173.95  , -180 , 0 , 90];
	aPosePassedSmallSt4			: ARRAY [1..6] OF REAL := [-72.2, 189.4545 ,173.95  , -180 , 0 , 90];
	
	rLinPosPalletPass : LREAL; // Linear axis position for placing passed assembly for selected station
	rLinPosPalletReject : LREAL; // Linear axis position for placing rejected assembly for selected station
	
END_STRUCT
END_TYPE

// ---- POUs/Meca500/Op/PoseData/ST_Sts2_PoseData.TcDUT
TYPE ST_Sts2_PoseData :
STRUCT
	
	aPoseSmallMotorPickupSt1 : ARRAY [1..6] OF REAL := [-222.713, 67.9 , 150, 180, -20 ,0] ; // Pose before gripper in to the pallet picking position
	aPoseSmallMotorPickupSt2 : ARRAY [1..6] OF REAL := [-222.713, 67.9 , 112.2, 180, -20 ,0] ; // Pose before gripper grip, or pose after gripper grip
	aPoseSmallMotorPickupSt3 : ARRAY [1..6] OF REAL := [-220.552, 67.9 , 111.4134, 180, -20 ,0] ; // Pose gripper grip
	rLinPosSmallMotorPickup				: LREAL := 80; // Linear axis position for pickup functions for selected station
	
	aPoseSmallMotorPlaceSt1 : ARRAY [1..6] OF REAL := [-144.652, 129 , 110.5 , 0, -90 ,0] ; // Pose before Small motor in station
	aPoseSmallMotorPlaceSt2 : ARRAY [1..6] OF REAL  := [-224.652, 129 , 110.5 , 0, -90 ,0]; // Pose Small motor in station
	rLinPosPlace : LREAL := 10; // Linear axis position for placing functions for selected station

	aPoseMirrorAdj : ARRAY[1..6] OF REAL; // Pose where final position of left mirror is saved in case position adjustment is needed.
	
	aPoseLargeMotorPickupSt1	: ARRAY [1..6] OF REAL := [-124.609, 117.800 , 101.6 , 0, -90 ,0]; // POSE BEFORE ACTUAL GRIP POSITION -108.2
	aPoseLargeMotorPickupSt2	: ARRAY [1..6] OF REAL := [-224.609, 117.800 , 101.6 , 0, -90 ,0];// ACTUAL GRIP POSITION
	aPoseLargeMotorPickupSt3	: ARRAY [1..6] OF REAL := [-224.609, 117.800 , 201.6 , 0, -90 ,0];// MOTOR LIFT FROM PALLET
	rLinPosMotorPickup				: LREAL := 160; // Linear axis position for pickup functions for selected station
	
	aPoseLargeMotorPlaceSt1	: ARRAY [1..6] OF REAL := [27.350, 79.603 , 67.4 , 180, 0 ,90]; // POSE BEFORE ACTULA LEAVING POSITION '
	aPoseLargeMotorPlaceSt2	: ARRAY [1..6] OF REAL := [27.350, 145.603 , 67.4 , 180, 0 ,90]; // ACTUAL POSITION FOR LEAVING MOTOR AT CURING STATION '
	aPoseLargeMotorPlaceSt3	: ARRAY [1..6] OF REAL := [27.350, 145.603 , 100.6 , 180, 0 ,90]; // POSE AFTER LEAVING MOTOR AT CURING STATION '
	
	aPoseMirrorPickupSt1	: ARRAY [1..6] OF REAL := [-158.94, 76.3 , 120, 181, 0 ,0]; // POSE BEFORE ACTUAL GRIP POSITION
	aPoseMirrorPickupSt2	: ARRAY [1..6] OF REAL := [-158.94, 76.3 , 81.55, 181, 0 ,0];// ACTUAL GRIP POSITION 187.1757
	rLinPosMirrorPickup				: LREAL := 137; // Linear axis position for pickup functions for selected station
	
// 	aPoseG14MirrorPlaceSt1	: ARRAY [1..6] OF REAL := [-72, 190.6 ,117.4 , 180, 0 ,90]; // POSE BEFORE INSERTIN MIRROR IN STATION'
// 	aPoseG14MirrorPlaceSt2	: ARRAY [1..6] OF REAL := [-72, 188.2 ,70.4 , -170, 0 ,90]; // POSE MIRROR IN STATION BUT NOT INSERTED TO MOTOR '
// 	aPoseg14MirrorPlaceSt3	: ARRAY [1..6] OF REAL := [-72, 187 ,68.6 , -180, 0 ,90]; // POSE MIRROR INSERTED TO MOTOR'
	
	aPoseG14MirrorPlaceSt1	: ARRAY [1..6] OF REAL := [27.350, 190.66 ,117.4 , 180, 0 ,90]; // POSE BEFORE INSERTIN MIRROR IN STATION'
	aPoseG14MirrorPlaceSt2	: ARRAY [1..6] OF REAL := [27.350, 191.66 ,70.4 , -170, 0 ,90]; // POSE MIRROR IN STATION BUT NOT INSERTED TO MOTOR '
	aPoseg14MirrorPlaceSt3	: ARRAY [1..6] OF REAL := [27.350, 190.16 ,68.6 , -178.5, -0.2 ,90]; // POSE MIRROR INSERTED TO MOTOR'
	
	aPosePassedLargeSt1 		: ARRAY [1..6] OF REAL := [-213.4, 62.25 , 141.45, 180, -20 ,0]; // In and out of pallet
	aPosePassedLargeSt2			: ARRAY [1..6] OF REAL := [-223.4, 62.25 , 101.45, 180, -20 ,0]; // before leaving position
	aPosePassedLargeSt3			: ARRAY [1..6] OF REAL := [-228, 62.25 ,97.79, 180, -20 ,0]; // Leaving position
	
	aPosePassedSmallSt1			: ARRAY [1..6] OF REAL := [-72.2, 189.4545 ,173.95  , -180 , 0 , 90];
	aPosePassedSmallSt2			: ARRAY [1..6] OF REAL := [-72.2, 189.4545 ,173.95  , -180 , 0 , 90];
	aPosePassedSmallSt3			: ARRAY [1..6] OF REAL := [-72.2, 189.4545 ,173.95  , -180 , 0 , 90];
	aPosePassedSmallSt4			: ARRAY [1..6] OF REAL := [-72.2, 189.4545 ,173.95  , -180 , 0 , 90];
	
	rLinPosPalletPass : LREAL := 320; // Linear axis position for placing passed assembly for selected station
	rLinPosPalletReject : LREAL; // Linear axis position for placing rejected assembly for selected station
	
END_STRUCT
END_TYPE

// ---- POUs/Meca500/Op/PoseData/ST_Sts3_PoseData.TcDUT
TYPE ST_Sts3_PoseData :
STRUCT
	
	aPoseSmallMotorPickupSt1 : ARRAY [1..6] OF REAL := [-222.713, 67.9 , 150, 180, -20 ,0] ; // Pose before gripper in to the pallet picking position
	aPoseSmallMotorPickupSt2 : ARRAY [1..6] OF REAL := [-222.713, 67.9 , 112.2, 180, -20 ,0] ; // Pose before gripper grip, or pose after gripper grip
	aPoseSmallMotorPickupSt3 : ARRAY [1..6] OF REAL := [-220.552, 67.9 , 111.4134, 180, -20 ,0] ; // Pose gripper grip
	rLinPosSmallMotorPickup				: LREAL := 80; // Linear axis position for pickup functions for selected station
	
	aPoseSmallMotorPlaceSt1 : ARRAY [1..6] OF REAL := [-144.652, 129 , 110.5 , 0, -90 ,0] ; // Pose before Small motor in station
	aPoseSmallMotorPlaceSt2 : ARRAY [1..6] OF REAL  := [-224.652, 129 , 110.5 , 0, -90 ,0]; // Pose Small motor in station
	rLinPosPlace : LREAL := 10; // Linear axis position for placing functions for selected station

	aPoseMirrorAdj : ARRAY[1..6] OF REAL; // Pose where final position of left mirror is saved in case position adjustment is needed.
	
	aPoseLargeMotorPickupSt1	: ARRAY [1..6] OF REAL := [-124.609, 117.800 , 101.6 , 0, -90 ,0]; // POSE BEFORE ACTUAL GRIP POSITION -108.2
	aPoseLargeMotorPickupSt2	: ARRAY [1..6] OF REAL := [-224.609, 117.800 , 101.6 , 0, -90 ,0];// ACTUAL GRIP POSITION
	aPoseLargeMotorPickupSt3	: ARRAY [1..6] OF REAL := [-224.609, 117.800 , 201.6 , 0, -90 ,0];// MOTOR LIFT FROM PALLET
	rLinPosMotorPickup				: LREAL := 160; // Linear axis position for pickup functions for selected station
	
	aPoseLargeMotorPlaceSt1	: ARRAY [1..6] OF REAL := [27.350, 79.603 , 67.4 , 180, 0 ,90]; // POSE BEFORE ACTULA LEAVING POSITION '
	aPoseLargeMotorPlaceSt2	: ARRAY [1..6] OF REAL := [27.350, 145.603 , 67.4 , 180, 0 ,90]; // ACTUAL POSITION FOR LEAVING MOTOR AT CURING STATION '
	aPoseLargeMotorPlaceSt3	: ARRAY [1..6] OF REAL := [27.350, 145.603 , 100.6 , 180, 0 ,90]; // POSE AFTER LEAVING MOTOR AT CURING STATION '
	
	aPoseMirrorPickupSt1	: ARRAY [1..6] OF REAL := [-173.9, 76.3 , 120, 181, 0 ,0]; // POSE BEFORE ACTUAL GRIP POSITION
	aPoseMirrorPickupSt2	: ARRAY [1..6] OF REAL := [-173.9, 76.3 , 81.55, 181, 0 ,0];// ACTUAL GRIP POSITION 187.1757
	rLinPosMirrorPickup				: LREAL := 108.625; // Linear axis position for pickup functions for selected station
	
// 	aPoseG14MirrorPlaceSt1	: ARRAY [1..6] OF REAL := [-72, 190.6 ,117.4 , 180, 0 ,90]; // POSE BEFORE INSERTIN MIRROR IN STATION'
// 	aPoseG14MirrorPlaceSt2	: ARRAY [1..6] OF REAL := [-72, 188.2 ,70.4 , -170, 0 ,90]; // POSE MIRROR IN STATION BUT NOT INSERTED TO MOTOR '
// 	aPoseg14MirrorPlaceSt3	: ARRAY [1..6] OF REAL := [-72, 187 ,68.6 , -180, 0 ,90]; // POSE MIRROR INSERTED TO MOTOR'
	
	aPoseG14MirrorPlaceSt1	: ARRAY [1..6] OF REAL := [27.350, 190.66 ,117.4 , 180, 0 ,90]; // POSE BEFORE INSERTIN MIRROR IN STATION'
	aPoseG14MirrorPlaceSt2	: ARRAY [1..6] OF REAL := [27.350, 191.66 ,70.4 , -170, 0 ,90]; // POSE MIRROR IN STATION BUT NOT INSERTED TO MOTOR '
	aPoseg14MirrorPlaceSt3	: ARRAY [1..6] OF REAL := [27.350, 190.16 ,68.6 , -178.5, -0.2 ,90]; // POSE MIRROR INSERTED TO MOTOR'
	
	aPosePassedLargeSt1 		: ARRAY [1..6] OF REAL := [-213.4, 62.25 , 141.45, 180, -20 ,0]; // In and out of pallet
	aPosePassedLargeSt2			: ARRAY [1..6] OF REAL := [-223.4, 62.25 , 101.45, 180, -20 ,0]; // before leaving position
	aPosePassedLargeSt3			: ARRAY [1..6] OF REAL := [-228, 62.25 ,97.79, 180, -20 ,0]; // Leaving position
	
	aPosePassedSmallSt1			: ARRAY [1..6] OF REAL := [-72.2, 189.4545 ,173.95  , -180 , 0 , 90];
	aPosePassedSmallSt2			: ARRAY [1..6] OF REAL := [-72.2, 189.4545 ,173.95  , -180 , 0 , 90];
	aPosePassedSmallSt3			: ARRAY [1..6] OF REAL := [-72.2, 189.4545 ,173.95  , -180 , 0 , 90];
	aPosePassedSmallSt4			: ARRAY [1..6] OF REAL := [-72.2, 189.4545 ,173.95  , -180 , 0 , 90];
	
	rLinPosPalletPass : LREAL := 320; // Linear axis position for placing passed assembly for selected station
	rLinPosPalletReject : LREAL; // Linear axis position for placing rejected assembly for selected station
	
END_STRUCT
END_TYPE

// ---- POUs/Meca500/Op/PoseData/ST_Sts4_PoseData.TcDUT
TYPE ST_Sts4_PoseData :
STRUCT
	
	aPoseSmallMotorPickupSt1 : ARRAY [1..6] OF REAL := [-222.713, 67.9 , 150, 180, -20 ,0] ; // Pose before gripper in to the pallet picking position
	aPoseSmallMotorPickupSt2 : ARRAY [1..6] OF REAL := [-222.713, 67.9 , 112.2, 180, -20 ,0] ; // Pose before gripper grip, or pose after gripper grip
	aPoseSmallMotorPickupSt3 : ARRAY [1..6] OF REAL := [-220.552, 67.9 , 111.4134, 180, -20 ,0] ; // Pose gripper grip
	rLinPosSmallMotorPickup				: LREAL := 80; // Linear axis position for pickup functions for selected station
	
	aPoseSmallMotorPlaceSt1 : ARRAY [1..6] OF REAL := [-144.652, 129 , 110.5 , 0, -90 ,0] ; // Pose before Small motor in station
	aPoseSmallMotorPlaceSt2 : ARRAY [1..6] OF REAL  := [-224.652, 129 , 110.5 , 0, -90 ,0]; // Pose Small motor in station
	rLinPosPlace : LREAL := 10; // Linear axis position for placing functions for selected station

	aPoseMirrorAdj : ARRAY[1..6] OF REAL; // Pose where final position of left mirror is saved in case position adjustment is needed.
	
	aPoseLargeMotorPickupSt1	: ARRAY [1..6] OF REAL := [-124.609, 117.800 , 101.6 , 0, -90 ,0]; // POSE BEFORE ACTUAL GRIP POSITION -108.2
	aPoseLargeMotorPickupSt2	: ARRAY [1..6] OF REAL := [-224.609, 117.800 , 101.6 , 0, -90 ,0];// ACTUAL GRIP POSITION
	aPoseLargeMotorPickupSt3	: ARRAY [1..6] OF REAL := [-224.609, 117.800 , 201.6 , 0, -90 ,0];// MOTOR LIFT FROM PALLET
	rLinPosMotorPickup				: LREAL := 120; // Linear axis position for pickup functions for selected station
	
	aPoseLargeMotorPlaceSt1	: ARRAY [1..6] OF REAL := [-73.3, 80 , 67.6 , 180, 0 ,90]; // POSE BEFORE ACTULA LEAVING POSITION '
	aPoseLargeMotorPlaceSt2	: ARRAY [1..6] OF REAL := [-73.3, 146 , 67.6 , 180, 0 ,90]; // ACTUAL POSITION FOR LEAVING MOTOR AT CURING STATION '
	aPoseLargeMotorPlaceSt3	: ARRAY [1..6] OF REAL := [-73.3, 146 , 100.6 , 180, 0 ,90]; // POSE AFTER LEAVING MOTOR AT CURING STATION '
	
	aPoseMirrorPickupSt1	: ARRAY [1..6] OF REAL := [-188.84, 76.3 , 120, 181, 0 ,0]; // POSE BEFORE ACTUAL GRIP POSITION
	aPoseMirrorPickupSt2	: ARRAY [1..6] OF REAL := [-188.84, 76.3 , 81.55, 181, 0 ,0];// ACTUAL GRIP POSITION 187.1757
	rLinPosMirrorPickup				: LREAL := 80; // Linear axis position for pickup functions for selected station
	
// 	aPoseG14MirrorPlaceSt1	: ARRAY [1..6] OF REAL := [-72, 190.6 ,117.4 , 180, 0 ,90]; // POSE BEFORE INSERTIN MIRROR IN STATION'
// 	aPoseG14MirrorPlaceSt2	: ARRAY [1..6] OF REAL := [-72, 188.2 ,70.4 , -170, 0 ,90]; // POSE MIRROR IN STATION BUT NOT INSERTED TO MOTOR '
// 	aPoseg14MirrorPlaceSt3	: ARRAY [1..6] OF REAL := [-72, 187 ,68.6 , -180, 0 ,90]; // POSE MIRROR INSERTED TO MOTOR'
	
	aPoseG14MirrorPlaceSt1	: ARRAY [1..6] OF REAL := [-73.3, 190.6 ,117.4 , 180, 0 ,90]; // POSE BEFORE INSERTIN MIRROR IN STATION'
	aPoseG14MirrorPlaceSt2	: ARRAY [1..6] OF REAL := [-73.3, 191.6 ,70.4 , -170, 0 ,90]; // POSE MIRROR IN STATION BUT NOT INSERTED TO MOTOR '
	aPoseg14MirrorPlaceSt3	: ARRAY [1..6] OF REAL := [-73.3, 190.1 ,68.6 , -178.5, -0.2 ,90]; // POSE MIRROR INSERTED TO MOTOR'
	
	aPosePassedLargeSt1 		: ARRAY [1..6] OF REAL := [-213.4, 62.25 , 141.45, 180, -20 ,0]; // In and out of pallet
	aPosePassedLargeSt2			: ARRAY [1..6] OF REAL := [-223.4, 62.25 , 101.45, 180, -20 ,0]; // before leaving position
	aPosePassedLargeSt3			: ARRAY [1..6] OF REAL := [-228, 62.25 ,97.79, 180, -20 ,0]; // Leaving position
	
	aPosePassedSmallSt1			: ARRAY [1..6] OF REAL := [-72.2, 189.4545 ,173.95  , -180 , 0 , 90];
	aPosePassedSmallSt2			: ARRAY [1..6] OF REAL := [-72.2, 189.4545 ,173.95  , -180 , 0 , 90];
	aPosePassedSmallSt3			: ARRAY [1..6] OF REAL := [-72.2, 189.4545 ,173.95  , -180 , 0 , 90];
	aPosePassedSmallSt4			: ARRAY [1..6] OF REAL := [-72.2, 189.4545 ,173.95  , -180 , 0 , 90];
	
	rLinPosPalletPass : LREAL := 280; // Linear axis position for placing passed assembly for selected station
	rLinPosPalletReject : LREAL; // Linear axis position for placing rejected assembly for selected station
	
END_STRUCT
END_TYPE

// ---- POUs/Meca500/Op/PoseData/ST_Sts5_PoseData.TcDUT
TYPE ST_Sts5_PoseData :
STRUCT
	
	aPoseSmallMotorPlaceSt1 : ARRAY [1..6] OF REAL; // Pose before Small motor in station
	aPoseSmallMotorPlaceSt2 : ARRAY [1..6] OF REAL; // Pose Small motor in station
	rLinPosPlace : LREAL; // Linear axis position for placing functions for selected station

	aPoseMirrorAdj : ARRAY[1..6] OF REAL; // Pose where final position of left mirror is saved in case position adjustment is needed.
	
	aPoseLargeMotorPickupSt1	: ARRAY [1..6] OF REAL := [-95,-150.45 , 110.5 , 0, -90 ,0]; // POSE BEFORE ACTUAL GRIP POSITION -108.2
	aPoseLargeMotorPickupSt2	: ARRAY [1..6] OF REAL := [-128.2,-150.45 , 110.5 , 0, -90 ,0];// ACTUAL GRIP POSITION
	aPoseLargeMotorPickupSt3	: ARRAY [1..6] OF REAL := [-128.2,-150.45 , 200.5 , 0, -90 ,0];// MOTOR LIFT FROM PALLET
	rLinPosPickup				: LREAL; // Linear axis position for pickup functions for selected station
	
	aPoseLargeMotorPlaceSt1	: ARRAY [1..6] OF REAL := [-73.8605, 110 ,165.6645  , -180 , 0 , 90]; // POSE BEFORE ACTULA LEAVING POSITION
	aPoseLargeMotorPlaceSt2	: ARRAY [1..6] OF REAL := [-73.8605, 140 ,165.6645  , -180 , 0 , 90]; // ACTUAL POSITION FOR LEAVING MOTOR AT CURING STATION
	aPoseLargeMotorPlaceSt3	: ARRAY [1..6] OF REAL := [-73.8605, 140 ,200  , -180 , 0 , 90]; // POSE AFTER LEAVING MOTOR AT CURING STATION
	
	aPoseMirrorPickupSt1	: ARRAY [1..6] OF REAL := [-159.1,-91.5 , 200 ,180, 0 ,0]; // POSE BEFORE ACTUAL GRIP POSITION
	aPoseMirrorPickupSt2	: ARRAY [1..6] OF REAL := [-159.1,-91.5 , 186.9757 ,180, 0 ,0];// ACTUAL GRIP POSITION 187.1757
	
	aPoseMirrorPlaceSt1	: ARRAY [1..6] OF REAL := [-72.2, 192.8 ,200.3  , -180 , 0 , 90]; // POSE BEFORE INSERTIN MIRROR IN STATION
	aPoseMirrorPlaceSt2	: ARRAY [1..6] OF REAL := [-72.2, 192.8 ,173.55  , -180 , 0 , 90]; // POSE MIRROR IN STATION BUT NOT INSERTED TO MOTOR  192.8, 173.45
	aPoseMirrorPlaceSt3	: ARRAY [1..6] OF REAL := [-72.2, 189.4545 ,173.95  , -180 , 0 , 90]; // POSE MIRROR INSERTED TO MOTOR
	
	aPosePassedLargeSt1 		: ARRAY [1..6] OF REAL := [-72.2, 189.4545 ,173.95  , -180 , 0 , 90];
	aPosePassedLargeSt2			: ARRAY [1..6] OF REAL := [-72.2, 189.4545 ,173.95  , -180 , 0 , 90];
	aPosePassedLargeSt3			: ARRAY [1..6] OF REAL := [-72.2, 189.4545 ,173.95  , -180 , 0 , 90];
	
	aPosePassedSmallSt1			: ARRAY [1..6] OF REAL := [-72.2, 189.4545 ,173.95  , -180 , 0 , 90];
	aPosePassedSmallSt2			: ARRAY [1..6] OF REAL := [-72.2, 189.4545 ,173.95  , -180 , 0 , 90];
	aPosePassedSmallSt3			: ARRAY [1..6] OF REAL := [-72.2, 189.4545 ,173.95  , -180 , 0 , 90];
	aPosePassedSmallSt4			: ARRAY [1..6] OF REAL := [-72.2, 189.4545 ,173.95  , -180 , 0 , 90];
	
	rLinPosPalletPass : LREAL; // Linear axis position for placing passed assembly for selected station
	rLinPosPalletReject : LREAL; // Linear axis position for placing rejected assembly for selected station
	
END_STRUCT
END_TYPE

// ---- POUs/Meca500/Op/PoseData/ST_Sts6_PoseData.TcDUT
TYPE ST_Sts6_PoseData :
STRUCT
	
	aPoseSmallMotorPlaceSt1 : ARRAY [1..6] OF REAL; // Pose before Small motor in station
	aPoseSmallMotorPlaceSt2 : ARRAY [1..6] OF REAL; // Pose Small motor in station
	rLinPosPlace : LREAL; // Linear axis position for placing functions for selected station

	aPoseMirrorAdj : ARRAY[1..6] OF REAL; // Pose where final position of left mirror is saved in case position adjustment is needed.
	
	aPoseLargeMotorPickupSt1	: ARRAY [1..6] OF REAL := [-95,-150.45 , 110.5 , 0, -90 ,0]; // POSE BEFORE ACTUAL GRIP POSITION -108.2
	aPoseLargeMotorPickupSt2	: ARRAY [1..6] OF REAL := [-128.2,-150.45 , 110.5 , 0, -90 ,0];// ACTUAL GRIP POSITION
	aPoseLargeMotorPickupSt3	: ARRAY [1..6] OF REAL := [-128.2,-150.45 , 200.5 , 0, -90 ,0];// MOTOR LIFT FROM PALLET
	rLinPosPickup				: LREAL; // Linear axis position for pickup functions for selected station
	
	aPoseLargeMotorPlaceSt1	: ARRAY [1..6] OF REAL := [-73.8605, 110 ,165.6645  , -180 , 0 , 90]; // POSE BEFORE ACTULA LEAVING POSITION
	aPoseLargeMotorPlaceSt2	: ARRAY [1..6] OF REAL := [-73.8605, 140 ,165.6645  , -180 , 0 , 90]; // ACTUAL POSITION FOR LEAVING MOTOR AT CURING STATION
	aPoseLargeMotorPlaceSt3	: ARRAY [1..6] OF REAL := [-73.8605, 140 ,200  , -180 , 0 , 90]; // POSE AFTER LEAVING MOTOR AT CURING STATION
	
	aPoseMirrorPickupSt1	: ARRAY [1..6] OF REAL := [-159.1,-91.5 , 200 ,180, 0 ,0]; // POSE BEFORE ACTUAL GRIP POSITION
	aPoseMirrorPickupSt2	: ARRAY [1..6] OF REAL := [-159.1,-91.5 , 186.9757 ,180, 0 ,0];// ACTUAL GRIP POSITION 187.1757
	
	aPoseMirrorPlaceSt1	: ARRAY [1..6] OF REAL := [-72.2, 192.8 ,200.3  , -180 , 0 , 90]; // POSE BEFORE INSERTIN MIRROR IN STATION
	aPoseMirrorPlaceSt2	: ARRAY [1..6] OF REAL := [-72.2, 192.8 ,173.55  , -180 , 0 , 90]; // POSE MIRROR IN STATION BUT NOT INSERTED TO MOTOR  192.8, 173.45
	aPoseMirrorPlaceSt3	: ARRAY [1..6] OF REAL := [-72.2, 189.4545 ,173.95  , -180 , 0 , 90]; // POSE MIRROR INSERTED TO MOTOR
	
	aPosePassedLargeSt1 		: ARRAY [1..6] OF REAL := [-72.2, 189.4545 ,173.95  , -180 , 0 , 90];
	aPosePassedLargeSt2			: ARRAY [1..6] OF REAL := [-72.2, 189.4545 ,173.95  , -180 , 0 , 90];
	aPosePassedLargeSt3			: ARRAY [1..6] OF REAL := [-72.2, 189.4545 ,173.95  , -180 , 0 , 90];
	
	aPosePassedSmallSt1			: ARRAY [1..6] OF REAL := [-72.2, 189.4545 ,173.95  , -180 , 0 , 90];
	aPosePassedSmallSt2			: ARRAY [1..6] OF REAL := [-72.2, 189.4545 ,173.95  , -180 , 0 , 90];
	aPosePassedSmallSt3			: ARRAY [1..6] OF REAL := [-72.2, 189.4545 ,173.95  , -180 , 0 , 90];
	aPosePassedSmallSt4			: ARRAY [1..6] OF REAL := [-72.2, 189.4545 ,173.95  , -180 , 0 , 90];
	
	rLinPosPalletPass : LREAL; // Linear axis position for placing passed assembly for selected station
	rLinPosPalletReject : LREAL; // Linear axis position for placing rejected assembly for selected station
	
END_STRUCT
END_TYPE

// ---- POUs/Meca500/Op/PoseData/ST_Sts7_PoseData.TcDUT
TYPE ST_Sts7_PoseData :
STRUCT
	
	aPoseSmallMotorPlaceSt1 : ARRAY [1..6] OF REAL; // Pose before Small motor in station
	aPoseSmallMotorPlaceSt2 : ARRAY [1..6] OF REAL; // Pose Small motor in station
	rLinPosPlace : LREAL; // Linear axis position for placing functions for selected station

	aPoseMirrorAdj : ARRAY[1..6] OF REAL; // Pose where final position of left mirror is saved in case position adjustment is needed.
	
	aPoseLargeMotorPickupSt1	: ARRAY [1..6] OF REAL := [-95,-150.45 , 110.5 , 0, -90 ,0]; // POSE BEFORE ACTUAL GRIP POSITION -108.2
	aPoseLargeMotorPickupSt2	: ARRAY [1..6] OF REAL := [-128.2,-150.45 , 110.5 , 0, -90 ,0];// ACTUAL GRIP POSITION
	aPoseLargeMotorPickupSt3	: ARRAY [1..6] OF REAL := [-128.2,-150.45 , 200.5 , 0, -90 ,0];// MOTOR LIFT FROM PALLET
	rLinPosPickup				: LREAL; // Linear axis position for pickup functions for selected station
	
	aPoseLargeMotorPlaceSt1	: ARRAY [1..6] OF REAL := [-73.8605, 110 ,165.6645  , -180 , 0 , 90]; // POSE BEFORE ACTULA LEAVING POSITION
	aPoseLargeMotorPlaceSt2	: ARRAY [1..6] OF REAL := [-73.8605, 140 ,165.6645  , -180 , 0 , 90]; // ACTUAL POSITION FOR LEAVING MOTOR AT CURING STATION
	aPoseLargeMotorPlaceSt3	: ARRAY [1..6] OF REAL := [-73.8605, 140 ,200  , -180 , 0 , 90]; // POSE AFTER LEAVING MOTOR AT CURING STATION
	
	aPoseMirrorPickupSt1	: ARRAY [1..6] OF REAL := [-159.1,-91.5 , 200 ,180, 0 ,0]; // POSE BEFORE ACTUAL GRIP POSITION
	aPoseMirrorPickupSt2	: ARRAY [1..6] OF REAL := [-159.1,-91.5 , 186.9757 ,180, 0 ,0];// ACTUAL GRIP POSITION 187.1757
	
	aPoseMirrorPlaceSt1	: ARRAY [1..6] OF REAL := [-72.2, 192.8 ,200.3  , -180 , 0 , 90]; // POSE BEFORE INSERTIN MIRROR IN STATION
	aPoseMirrorPlaceSt2	: ARRAY [1..6] OF REAL := [-72.2, 192.8 ,173.55  , -180 , 0 , 90]; // POSE MIRROR IN STATION BUT NOT INSERTED TO MOTOR  192.8, 173.45
	aPoseMirrorPlaceSt3	: ARRAY [1..6] OF REAL := [-72.2, 189.4545 ,173.95  , -180 , 0 , 90]; // POSE MIRROR INSERTED TO MOTOR
	
	aPosePassedLargeSt1 		: ARRAY [1..6] OF REAL := [-72.2, 189.4545 ,173.95  , -180 , 0 , 90];
	aPosePassedLargeSt2			: ARRAY [1..6] OF REAL := [-72.2, 189.4545 ,173.95  , -180 , 0 , 90];
	aPosePassedLargeSt3			: ARRAY [1..6] OF REAL := [-72.2, 189.4545 ,173.95  , -180 , 0 , 90];
	
	aPosePassedSmallSt1			: ARRAY [1..6] OF REAL := [-72.2, 189.4545 ,173.95  , -180 , 0 , 90];
	aPosePassedSmallSt2			: ARRAY [1..6] OF REAL := [-72.2, 189.4545 ,173.95  , -180 , 0 , 90];
	aPosePassedSmallSt3			: ARRAY [1..6] OF REAL := [-72.2, 189.4545 ,173.95  , -180 , 0 , 90];
	aPosePassedSmallSt4			: ARRAY [1..6] OF REAL := [-72.2, 189.4545 ,173.95  , -180 , 0 , 90];
	
	rLinPosPalletPass : LREAL; // Linear axis position for placing passed assembly for selected station
	rLinPosPalletReject : LREAL; // Linear axis position for placing rejected assembly for selected station
	
END_STRUCT
END_TYPE

// ---- POUs/Meca500/Op/PoseData/ST_Sts8_PoseData.TcDUT
TYPE ST_Sts8_PoseData :
STRUCT
	
	aPoseSmallMotorPlaceSt1 : ARRAY [1..6] OF REAL; // Pose before Small motor in station
	aPoseSmallMotorPlaceSt2 : ARRAY [1..6] OF REAL; // Pose Small motor in station
	rLinPosPlace : LREAL; // Linear axis position for placing functions for selected station

	aPoseMirrorAdj : ARRAY[1..6] OF REAL; // Pose where final position of left mirror is saved in case position adjustment is needed.
	
	aPoseLargeMotorPickupSt1	: ARRAY [1..6] OF REAL := [-95,-150.45 , 110.5 , 0, -90 ,0]; // POSE BEFORE ACTUAL GRIP POSITION -108.2
	aPoseLargeMotorPickupSt2	: ARRAY [1..6] OF REAL := [-128.2,-150.45 , 110.5 , 0, -90 ,0];// ACTUAL GRIP POSITION
	aPoseLargeMotorPickupSt3	: ARRAY [1..6] OF REAL := [-128.2,-150.45 , 200.5 , 0, -90 ,0];// MOTOR LIFT FROM PALLET
	rLinPosPickup				: LREAL; // Linear axis position for pickup functions for selected station
	
	aPoseLargeMotorPlaceSt1	: ARRAY [1..6] OF REAL := [-73.8605, 110 ,165.6645  , -180 , 0 , 90]; // POSE BEFORE ACTULA LEAVING POSITION
	aPoseLargeMotorPlaceSt2	: ARRAY [1..6] OF REAL := [-73.8605, 140 ,165.6645  , -180 , 0 , 90]; // ACTUAL POSITION FOR LEAVING MOTOR AT CURING STATION
	aPoseLargeMotorPlaceSt3	: ARRAY [1..6] OF REAL := [-73.8605, 140 ,200  , -180 , 0 , 90]; // POSE AFTER LEAVING MOTOR AT CURING STATION
	
	aPoseMirrorPickupSt1	: ARRAY [1..6] OF REAL := [-159.1,-91.5 , 200 ,180, 0 ,0]; // POSE BEFORE ACTUAL GRIP POSITION
	aPoseMirrorPickupSt2	: ARRAY [1..6] OF REAL := [-159.1,-91.5 , 186.9757 ,180, 0 ,0];// ACTUAL GRIP POSITION 187.1757
	
	aPoseMirrorPlaceSt1	: ARRAY [1..6] OF REAL := [-72.2, 192.8 ,200.3  , -180 , 0 , 90]; // POSE BEFORE INSERTIN MIRROR IN STATION
	aPoseMirrorPlaceSt2	: ARRAY [1..6] OF REAL := [-72.2, 192.8 ,173.55  , -180 , 0 , 90]; // POSE MIRROR IN STATION BUT NOT INSERTED TO MOTOR  192.8, 173.45
	aPoseMirrorPlaceSt3	: ARRAY [1..6] OF REAL := [-72.2, 189.4545 ,173.95  , -180 , 0 , 90]; // POSE MIRROR INSERTED TO MOTOR
	
	aPosePassedLargeSt1 		: ARRAY [1..6] OF REAL := [-72.2, 189.4545 ,173.95  , -180 , 0 , 90];
	aPosePassedLargeSt2			: ARRAY [1..6] OF REAL := [-72.2, 189.4545 ,173.95  , -180 , 0 , 90];
	aPosePassedLargeSt3			: ARRAY [1..6] OF REAL := [-72.2, 189.4545 ,173.95  , -180 , 0 , 90];
	
	aPosePassedSmallSt1			: ARRAY [1..6] OF REAL := [-72.2, 189.4545 ,173.95  , -180 , 0 , 90];
	aPosePassedSmallSt2			: ARRAY [1..6] OF REAL := [-72.2, 189.4545 ,173.95  , -180 , 0 , 90];
	aPosePassedSmallSt3			: ARRAY [1..6] OF REAL := [-72.2, 189.4545 ,173.95  , -180 , 0 , 90];
	aPosePassedSmallSt4			: ARRAY [1..6] OF REAL := [-72.2, 189.4545 ,173.95  , -180 , 0 , 90];
	
	rLinPosPalletPass : LREAL; // Linear axis position for placing passed assembly for selected station
	rLinPosPalletReject : LREAL; // Linear axis position for placing rejected assembly for selected station
	
END_STRUCT
END_TYPE

// ---- POUs/Meca500/Op/PoseData/ST_Sts9_PoseData.TcDUT
TYPE ST_Sts9_PoseData :
STRUCT
	
	aPoseSmallMotorPlaceSt1 : ARRAY [1..6] OF REAL; // Pose before Small motor in station
	aPoseSmallMotorPlaceSt2 : ARRAY [1..6] OF REAL; // Pose Small motor in station
	rLinPosPlace : LREAL; // Linear axis position for placing functions for selected station

	aPoseMirrorAdj : ARRAY[1..6] OF REAL; // Pose where final position of left mirror is saved in case position adjustment is needed.
	
	aPoseLargeMotorPickupSt1	: ARRAY [1..6] OF REAL := [-95,-150.45 , 110.5 , 0, -90 ,0]; // POSE BEFORE ACTUAL GRIP POSITION -108.2
	aPoseLargeMotorPickupSt2	: ARRAY [1..6] OF REAL := [-128.2,-150.45 , 110.5 , 0, -90 ,0];// ACTUAL GRIP POSITION
	aPoseLargeMotorPickupSt3	: ARRAY [1..6] OF REAL := [-128.2,-150.45 , 200.5 , 0, -90 ,0];// MOTOR LIFT FROM PALLET
	rLinPosPickup				: LREAL; // Linear axis position for pickup functions for selected station
	
	aPoseLargeMotorPlaceSt1	: ARRAY [1..6] OF REAL := [-73.8605, 110 ,165.6645  , -180 , 0 , 90]; // POSE BEFORE ACTULA LEAVING POSITION
	aPoseLargeMotorPlaceSt2	: ARRAY [1..6] OF REAL := [-73.8605, 140 ,165.6645  , -180 , 0 , 90]; // ACTUAL POSITION FOR LEAVING MOTOR AT CURING STATION
	aPoseLargeMotorPlaceSt3	: ARRAY [1..6] OF REAL := [-73.8605, 140 ,200  , -180 , 0 , 90]; // POSE AFTER LEAVING MOTOR AT CURING STATION
	
	aPoseMirrorPickupSt1	: ARRAY [1..6] OF REAL := [-159.1,-91.5 , 200 ,180, 0 ,0]; // POSE BEFORE ACTUAL GRIP POSITION
	aPoseMirrorPickupSt2	: ARRAY [1..6] OF REAL := [-159.1,-91.5 , 186.9757 ,180, 0 ,0];// ACTUAL GRIP POSITION 187.1757
	
	aPoseMirrorPlaceSt1	: ARRAY [1..6] OF REAL := [-72.2, 192.8 ,200.3  , -180 , 0 , 90]; // POSE BEFORE INSERTIN MIRROR IN STATION
	aPoseMirrorPlaceSt2	: ARRAY [1..6] OF REAL := [-72.2, 192.8 ,173.55  , -180 , 0 , 90]; // POSE MIRROR IN STATION BUT NOT INSERTED TO MOTOR  192.8, 173.45
	aPoseMirrorPlaceSt3	: ARRAY [1..6] OF REAL := [-72.2, 189.4545 ,173.95  , -180 , 0 , 90]; // POSE MIRROR INSERTED TO MOTOR
	
	aPosePassedLargeSt1 		: ARRAY [1..6] OF REAL := [-72.2, 189.4545 ,173.95  , -180 , 0 , 90];
	aPosePassedLargeSt2			: ARRAY [1..6] OF REAL := [-72.2, 189.4545 ,173.95  , -180 , 0 , 90];
	aPosePassedLargeSt3			: ARRAY [1..6] OF REAL := [-72.2, 189.4545 ,173.95  , -180 , 0 , 90];
	
	aPosePassedSmallSt1			: ARRAY [1..6] OF REAL := [-72.2, 189.4545 ,173.95  , -180 , 0 , 90];
	aPosePassedSmallSt2			: ARRAY [1..6] OF REAL := [-72.2, 189.4545 ,173.95  , -180 , 0 , 90];
	aPosePassedSmallSt3			: ARRAY [1..6] OF REAL := [-72.2, 189.4545 ,173.95  , -180 , 0 , 90];
	aPosePassedSmallSt4			: ARRAY [1..6] OF REAL := [-72.2, 189.4545 ,173.95  , -180 , 0 , 90];
	
	rLinPosPalletPass : LREAL; // Linear axis position for placing passed assembly for selected station
	rLinPosPalletReject : LREAL; // Linear axis position for placing rejected assembly for selected station
	
END_STRUCT
END_TYPE

// ---- POUs/Meca500/Op/PoseData/Type/AL82027.TcDUT
TYPE AL82027 :
STRUCT
	PoseGluingSt1		:  ARRAY [1..6] OF REAL := [-185, 194 , 58.5 , -155, -10, 70]; // 
	PoseGluingSt2 		:  ARRAY [1..6] OF REAL := [-203.800, 209.037 , 64.824 , -110, -15, 90]; // 
	PoseGluingSt3 		:  ARRAY [1..6] OF REAL := [-200.238, 210.48 , 64.467 , -110, -15, 90]; // 
	PoseGluingSt4 		:  ARRAY [1..6] OF REAL := [-188.902, 190.264 , 80.928 , -155, -10, 70]; // 
// 	PoseGluingSt5		:  ARRAY [1..6] OF REAL := [-187.975, 194.011 , 82.274 , -155, -10, 70];  // 
	
// 	PoseGluingSt6 		:  ARRAY [1..6] OF REAL := [ -169.673813, 134.421356, 118.048595 , -123.6 , -17 , 90]; // 
// 	PoseGluingSt7 		:  ARRAY [1..6] OF REAL := [ -173.192612,132.9314, 118.355591 , -123.600 , -17 , 90];  //
// 	PoseGluingSt8		:  ARRAY [1..6] OF REAL := [ -174.150, 132.583 , 83.690 , -106.182 , -17 , 90];   //
// 	PoseGluingSt9		:  ARRAY [1..6] OF REAL := [ -169.879,134.182,83.645,-106.182,-17,90];  //
// 	PoseGluingSt10		:  ARRAY [1..6] OF REAL := [ -169.879,134.697,77,-106.182,-17,90];  //
	iPoseAmount			: INT := 4;
 	iGluingTimeLine			: INT := 5; // In Seconds
 	iGluingTimeDot			: INT := 5; // In Seconds
END_STRUCT
END_TYPE

// ---- POUs/Meca500/Op/PoseData/Type/AL86068.TcDUT
TYPE AL86068 :
STRUCT
	PoseGluingSt1		:  ARRAY [1..6] OF REAL := [-170.1, 134 ,165.7  , -167.5 , -4.7 , 72.5]; // 
	PoseGluingSt2 		:  ARRAY [1..6] OF REAL := [-175, 166 ,177.87  , -163.5 , -7.2 , 73.2]; // 
	PoseGluingSt3 		:  ARRAY [1..6] OF REAL := [-175, 166 ,160.27  , -163.5 , -7.2 , 73.2]; // 
	PoseGluingSt4 		:  ARRAY [1..6] OF REAL := [-157.9, 103.5 ,160.5  , -163.5 , -7.2 , 73.2]; // 
	PoseGluingSt5		:  ARRAY [1..6] OF REAL := [ -173.55, 132.8, 103 , -123.6 , -17 , 90];  // 
	
	PoseGluingSt6 		:  ARRAY [1..6] OF REAL := [ -169.673813, 134.421356, 118.048595 , -123.6 , -17 , 90]; // 
	PoseGluingSt7 		:  ARRAY [1..6] OF REAL := [ -173.192612,132.9314, 118.355591 , -123.600 , -17 , 90];  //
	PoseGluingSt8		:  ARRAY [1..6] OF REAL := [ -174.150, 132.583 , 83.690 , -106.182 , -17 , 90];   //
	PoseGluingSt9		:  ARRAY [1..6] OF REAL := [ -169.879,134.182,83.645,-106.182,-17,90];  //
	PoseGluingSt10		:  ARRAY [1..6] OF REAL := [ -169.879,134.697,77,-106.182,-17,90];  //
	iPoseAmount			: INT;
END_STRUCT
END_TYPE

// ---- POUs/Meca500/Op/PoseData/Type/AL200663.TcDUT
TYPE AL200663 :
STRUCT
	PoseGluingSt1		:  ARRAY [1..6] OF REAL := [-185, 194 , 58.5 , -155, -10, 70]; // 
	PoseGluingSt2 		:  ARRAY [1..6] OF REAL := [-190.946, 191.975 , 81.80 , -155.0, -10, 70]; // 
	PoseGluingSt3 		:  ARRAY [1..6] OF REAL := [-190.032, 189.277 , 80.544 , -155, -10, 70]; // 
	PoseGluingSt4 		:  ARRAY [1..6] OF REAL := [-186.869, 190.908 , 80.344 , -155, -10, 70]; // 
	PoseGluingSt5		:  ARRAY [1..6] OF REAL := [-187.975, 194.011 , 81.774 , -155, -10, 70];  // 
	
// 	PoseGluingSt6 		:  ARRAY [1..6] OF REAL := [ -169.673813, 134.421356, 118.048595 , -123.6 , -17 , 90]; // 
// 	PoseGluingSt7 		:  ARRAY [1..6] OF REAL := [ -173.192612,132.9314, 118.355591 , -123.600 , -17 , 90];  //
// 	PoseGluingSt8		:  ARRAY [1..6] OF REAL := [ -174.150, 132.583 , 83.690 , -106.182 , -17 , 90];   //
// 	PoseGluingSt9		:  ARRAY [1..6] OF REAL := [ -169.879,134.182,83.645,-106.182,-17,90];  //
// 	PoseGluingSt10		:  ARRAY [1..6] OF REAL := [ -169.879,134.697,77,-106.182,-17,90];  //
	iPoseAmount			: INT := 5;
	iGluingTime			: INT := 5; // In Seconds
END_STRUCT
END_TYPE

// ---- POUs/Meca500/Op/PoseData/Type/AL200665.TcDUT
TYPE AL200665 :
STRUCT
	PoseGluingSt1		:  ARRAY [1..6] OF REAL := [-185, 194 , 58.5 , -155, -10, 70]; // 
	PoseGluingSt2 		:  ARRAY [1..6] OF REAL := [-190.946, 191.975 , 81.80 , -155.0, -10, 70]; // 
	PoseGluingSt3 		:  ARRAY [1..6] OF REAL := [-190.032, 189.277 , 80.544 , -155, -10, 70]; // 
	PoseGluingSt4 		:  ARRAY [1..6] OF REAL := [-186.869, 190.908 , 80.344 , -155, -10, 70]; // 
	PoseGluingSt5		:  ARRAY [1..6] OF REAL := [-187.975, 194.011 , 81.774 , -155, -10, 70];  // 
	
// 	PoseGluingSt6 		:  ARRAY [1..6] OF REAL := [ -169.673813, 134.421356, 118.048595 , -123.6 , -17 , 90]; // 
// 	PoseGluingSt7 		:  ARRAY [1..6] OF REAL := [ -173.192612,132.9314, 118.355591 , -123.600 , -17 , 90];  //
// 	PoseGluingSt8		:  ARRAY [1..6] OF REAL := [ -174.150, 132.583 , 83.690 , -106.182 , -17 , 90];   //
// 	PoseGluingSt9		:  ARRAY [1..6] OF REAL := [ -169.879,134.182,83.645,-106.182,-17,90];  //
// 	PoseGluingSt10		:  ARRAY [1..6] OF REAL := [ -169.879,134.697,77,-106.182,-17,90];  //
	iPoseAmount			: INT := 5;
	iGluingTime			: INT := 5; // In Seconds
END_STRUCT
END_TYPE

// ---- POUs/Meca500/Op/PoseData/Type/AL200664.TcDUT
TYPE AL200664 :
STRUCT
	PoseGluingSt1		:  ARRAY [1..6] OF REAL := [-185, 194 , 58.5 , -155, -10, 70]; // 
	PoseGluingSt2 		:  ARRAY [1..6] OF REAL := [-190.946, 191.975 , 82.30 , -155.0, -10, 70]; // 
	PoseGluingSt3 		:  ARRAY [1..6] OF REAL := [-190.032, 189.277 , 81.044 , -155, -10, 70]; // 
	PoseGluingSt4 		:  ARRAY [1..6] OF REAL := [-186.869, 190.908 , 80.844 , -155, -10, 70]; // 
	PoseGluingSt5		:  ARRAY [1..6] OF REAL := [-187.975, 194.011 , 82.274 , -155, -10, 70];  // 
	
// 	PoseGluingSt6 		:  ARRAY [1..6] OF REAL := [ -169.673813, 134.421356, 118.048595 , -123.6 , -17 , 90]; // 
// 	PoseGluingSt7 		:  ARRAY [1..6] OF REAL := [ -173.192612,132.9314, 118.355591 , -123.600 , -17 , 90];  //
// 	PoseGluingSt8		:  ARRAY [1..6] OF REAL := [ -174.150, 132.583 , 83.690 , -106.182 , -17 , 90];   //
// 	PoseGluingSt9		:  ARRAY [1..6] OF REAL := [ -169.879,134.182,83.645,-106.182,-17,90];  //
// 	PoseGluingSt10		:  ARRAY [1..6] OF REAL := [ -169.879,134.697,77,-106.182,-17,90];  //
	iPoseAmount			: INT := 5;
	iGluingTime			: INT := 5; // In Seconds
END_STRUCT
END_TYPE

// ---- POUs/Meca500/Op/PoseData/Type/AL200662.TcDUT
TYPE AL200662 :
STRUCT
	PoseGluingSt1		:  ARRAY [1..6] OF REAL := [-185, 194 , 58.5 , -155, -10, 70]; // 
	PoseGluingSt2 		:  ARRAY [1..6] OF REAL := [-190.946, 191.975 , 82.30 , -155.0, -10, 70]; // 
	PoseGluingSt3 		:  ARRAY [1..6] OF REAL := [-190.032, 189.277 , 81.044 , -155, -10, 70]; // 
	PoseGluingSt4 		:  ARRAY [1..6] OF REAL := [-186.869, 190.908 , 80.844 , -155, -10, 70]; // 
	PoseGluingSt5		:  ARRAY [1..6] OF REAL := [-187.975, 194.011 , 82.274 , -155, -10, 70];  // 
	
// 	PoseGluingSt6 		:  ARRAY [1..6] OF REAL := [ -169.673813, 134.421356, 118.048595 , -123.6 , -17 , 90]; // 
// 	PoseGluingSt7 		:  ARRAY [1..6] OF REAL := [ -173.192612,132.9314, 118.355591 , -123.600 , -17 , 90];  //
// 	PoseGluingSt8		:  ARRAY [1..6] OF REAL := [ -174.150, 132.583 , 83.690 , -106.182 , -17 , 90];   //
// 	PoseGluingSt9		:  ARRAY [1..6] OF REAL := [ -169.879,134.182,83.645,-106.182,-17,90];  //
// 	PoseGluingSt10		:  ARRAY [1..6] OF REAL := [ -169.879,134.697,77,-106.182,-17,90];  //
	iPoseAmount			: INT := 5;
	iGluingTime			: INT := 5; // In Seconds
END_STRUCT
END_TYPE

// ---- POUs/Sts/Com/ST_Stations.TcDUT
TYPE ST_Stations :
STRUCT
	fbSts1		: FB_StsAct;
	fbSts2		: FB_StsAct;
	fbSts3		: FB_StsAct;
	fbSts4		: FB_StsAct;
	fbSts5		: FB_StsAct;
	fbSts6		: FB_StsAct;
	fbSts7		: FB_StsAct;
	fbSts8		: FB_StsAct;
	fbSts9		: FB_StsAct;
	fbSts10		: FB_StsAct;
	
	stSts1 : ST_Sts1_PoseData;
	stSts2 : ST_Sts2_PoseData;
	stSts3 : ST_Sts3_PoseData;
	stSts4 : ST_Sts4_PoseData;
	stSts5 : ST_Sts5_PoseData;
	stSts6 : ST_Sts6_PoseData;
	stSts7 : ST_Sts7_PoseData;
	stSts8 : ST_Sts8_PoseData;
	stSts9 : ST_Sts9_PoseData;
	stSts10 : ST_Sts10_PoseData;

END_STRUCT
END_TYPE

// ---- POUs/Sts/Com/ST_Sts_PlcCom.TcDUT
TYPE ST_Sts_PlcCom :
STRUCT
	
	stPlcComIn		AT %I*: ST_Sts_PlcComIn;
	stPlcComOut		AT %Q*: ST_Sts_PlcComOut;

END_STRUCT
END_TYPE

// ---- POUs/Sts/Com/ST_Sts_PlcComIn.TcDUT
TYPE ST_Sts_PlcComIn :
STRUCT
	bSliderHomeSensor		: BOOL;
	bAngleMotorSensor		: BOOL;
	bGripperHomeSensor		: BOOL;
	PtcRawTemp				: INT;
END_STRUCT
END_TYPE

// ---- POUs/Sts/Com/ST_Sts_PlcComOut.TcDUT
TYPE ST_Sts_PlcComOut :
STRUCT
	bUnderLight			: BOOL;
	bGripper			: BOOL;
	bPusher				: BOOL;
	bHeaterFan			: BOOL;
	bHeaterElement		: BOOL;
END_STRUCT
END_TYPE

// ---- POUs/Sts/Datalog/ST_LogEntry.TcDUT
TYPE ST_LogEntry :
STRUCT
    tStamp			: TIMESTRUCT;		//Ltime or time
    Var1   			: LREAL;
    Var2  			: LREAL;
    Var3			: INT;

END_STRUCT
END_TYPE

// ---- POUs/Sts/DUT/E_MovementState.TcDUT
{attribute 'qualified_only'}
{attribute 'strict'}
{attribute 'to_string'}
TYPE E_MovementState :
(
	Idle,
	Jog,
	Halt,
	Error,
	EncHoming,
	Home
	
);
END_TYPE

// ---- POUs/Sts/DUT/E_StepperState.TcDUT
TYPE E_StepperState :
	
(
	Offline,
	Reset,
	Power,
	Error,
	Operational,
	EncHoming,
	Homing,
	Jog
);

END_TYPE

// ---- POUs/Sts/DUT/E_StsActState.TcDUT
{attribute 'qualified_only'}
{attribute 'strict'}
{attribute 'to_string'}
TYPE E_StsActState :
(
	StartupCheck,
	AssemblyCheck,
	Idle,
	DataLogging,
	RobotSlotHold,
	AngleAdj,
	PositionAdj,
	ProductMounting,
	ProductDisMounting,
	Disabled,
	Error,
	HoldForValveRelease
);
END_TYPE

// ---- POUs/Sts/DUT/ST_AngleData.TcDUT
TYPE ST_AngleData :
STRUCT
	stLaserData1	: ST_Vis_Laser;
	stLaserData2	: ST_Vis_Laser;
	stLaserData3	: ST_Vis_Laser;
	stLaserData4	: ST_Vis_Laser;
	stLaserData5	: ST_Vis_Laser;
	stLaserData6	: ST_Vis_Laser;
	stLaserData7	: ST_Vis_Laser;
	stLaserData8	: ST_Vis_Laser;
	stLaserData9	: ST_Vis_Laser;
	stLaserData10	: ST_Vis_Laser;
	
END_STRUCT
END_TYPE

// ---- POUs/Sts/DUT/ST_Sts_DetectionData.TcDUT
TYPE ST_Sts_DetectionData :
STRUCT
	
	stLaser	: ST_Vis_Laser;
	stMirror : ST_Vis_Mirror;
	
END_STRUCT
END_TYPE

// ---- POUs/Sts/DUT/ST_Vis_Laser.TcDUT
TYPE ST_Vis_Laser :
STRUCT
	
	stLaserRectangle		: TcVnRotatedRectangle;
	rLaserOffsetToSetPoint	: ARRAY [0..1] OF LREAL;
	bImagingStatusOk		: BOOL;
	bImagingDone			: BOOL;
	bDetectionFailed		: BOOL;
	
END_STRUCT
END_TYPE

// ---- POUs/Sts/DUT/ST_Vis_Mirror.TcDUT
TYPE ST_Vis_Mirror :
STRUCT

	rDetectedMirrorTypeNumber	: ARRAY [0..10] OF LREAL;
	stMirrorRectangle			: TcVnRotatedRectangle;
	rMirrorOffsetToCalPoints 	: ARRAY [0..1] OF LREAL;
	rMirrorOffsetToMotor		: ARRAY [0..1] OF LREAL;
	bImagingStatusOk			: BOOL;
	bLightTestOk				: BOOL;
	bLaserTestOk				: BOOL;
	bDetectionFailed			: BOOL;
	bImagingDone				: BOOL;
	bReadyForTrigger			: BOOL;
	
END_STRUCT
END_TYPE

// ---- POUs/VisMain/ST_CouplerImagingData.TcDUT
TYPE ST_CouplerImagingData :
STRUCT
	bImagingDone	: BOOL;
	rCouplerAngleRad	: LREAL;
	rCouplerAngleDeg	: LREAL;
	bImageReceived : BOOL;
	bPartDetectFailed : BOOL;
	bPartDetectSucceeded	: BOOL;
END_STRUCT
END_TYPE

// ---- POUs/VisMain/ST_PalletImagingData.TcDUT
TYPE ST_PalletImagingData :
STRUCT
	bImagingDone : BOOL;
	bTogglePallet	: BOOL; // If true, Imaging is set to detect 10mm pallet
	bSuccess_10mmLocate : BOOL;
	bSuccess_14mmLocate : BOOL;
	bMirrorPalletImagingSucceeded : BOOL;
END_STRUCT
END_TYPE

// ---- GVLs/Color.TcGVL
{attribute 'qualified_only'}
VAR_GLOBAL
	Black	: TcVnVector4_LREAL := [0,0,0,0];
	White	: TcVnVector4_LREAL := [255,255,255,0];

	Maroon	: TcVnVector4_LREAL := [128,0,0,0];
	Red		: TcVnVector4_LREAL := [255,0,0,0];
	Orange	: TcVnVector4_LREAL := [255,165,0,0];
	Yellow	: TcVnVector4_LREAL := [255,255,0,0];
	Olive	: TcVnVector4_LREAL := [128,128,0,0];
	Green	: TcVnVector4_LREAL := [0,128,0,0];
	Purple	: TcVnVector4_LREAL := [128,0,128,0];
	Fuchsia	: TcVnVector4_LREAL := [255,0,255,0];
	Lime	: TcVnVector4_LREAL := [0,255,0,0];
	Teal	: TcVnVector4_LREAL := [0,128,128,0];
	Aqua	: TcVnVector4_LREAL := [0,255,255,0];
	Blue	: TcVnVector4_LREAL := [0,0,255,0];
	Navy	: TcVnVector4_LREAL := [0,0,128,0];
	Gray	: TcVnVector4_LREAL := [128,128,128,0];
	Silver	: TcVnVector4_LREAL := [192,192,192,0];

END_VAR

// ---- GVLs/Err.TcGVL
{attribute 'qualified_only'}
VAR_GLOBAL
	Err  : BOOL;
END_VAR

// ---- GVLs/Trig.TcGVL
{attribute 'qualified_only'}
VAR_GLOBAL	
	bMidStationCam	: BOOL;
	bInfeedCam		: BOOL;
	bOutfeedCam		: BOOL;
	bRejectCam		: BOOL;
	
	
END_VAR

// ---- POUs/HP/CURING_STATION/VISION/VISION_PARAMS.TcGVL
{attribute 'qualified_only'}
VAR_GLOBAL PERSISTENT
	couplerDetectParams:	ST_COUPLER_DETECT_SETTINGS;
END_VAR

// ---- POUs/HP/GVL/HEATER_CONTROL_SETTINGS.TcGVL
{attribute 'qualified_only'}
VAR_GLOBAL PERSISTENT
	{ attribute 'TcHmiSymbol.AddSymbol' }
	{ attribute 'TcHmiSymbol.ShowRecursively' }
	settings:	ST_CURING_STATION_HEATER_CONTROL_STATIC_SETTINGS;
END_VAR

// ---- POUs/HP/GVL/HMI.TcGVL
{attribute 'qualified_only'}
VAR_GLOBAL
	{ attribute 'TcHmiSymbol.AddSymbol' }
	{ attribute 'TcHmiSymbol.ShowRecursively' }
	curingStations:	ARRAY[0..4] OF ST_CURING_STATION_HMI;
	
	{ attribute 'TcHmiSymbol.AddSymbol' }
	{ attribute 'TcHmiSymbol.ShowRecursively' }
	cs:				ST_CS_HMI;
END_VAR

// ---- POUs/HP/GVL/MAIN_VISION_COMM_VARS.TcGVL
{attribute 'qualified_only'}
VAR_GLOBAL
END_VAR

// ---- POUs/HP/CURING_STATION/VISION/Coupler/I_ImageProcessor.TcIO
INTERFACE I_ImageProcessor

METHOD ic_cancelProcessing
VAR_INPUT
END_VAR
END_METHOD

METHOD ic_getCenterPoint : TcVnPoint2_REAL
END_METHOD

METHOD ic_process
VAR_INPUT
	iRawImage:			ITcVnImage;
	iProcessedImage:	ITcVnImage;
	iDisplayableImage:	ITcVnDisplayableImage;
END_VAR
END_METHOD

METHOD ic_processingError : BOOL
END_METHOD

METHOD ic_processingReady : BOOL
END_METHOD

END_INTERFACE

// ---- POUs/HP/CURING_STATION/VISION/Mirror/I_MirrorImageProcessor.TcIO
INTERFACE I_MirrorImageProcessor

METHOD ic_cancelProcessing
VAR_INPUT
END_VAR
END_METHOD

METHOD ic_getResult : REAL
END_METHOD

METHOD ic_process
VAR_INPUT
	iRawImage:			ITcVnImage;
	iProcessedImage:	ITcVnImage;
	iDisplayableImage:	ITcVnDisplayableImage;
	iCameraPtr:			POINTER TO FB_VN_GevCameraControl;
	iCouplerCenterPoint:	TcVnPoint2_REAL;	
END_VAR
END_METHOD

METHOD ic_processingError : BOOL
END_METHOD

METHOD ic_processingReady : BOOL
END_METHOD

END_INTERFACE

// ---- POUs/MAIN.TcPOU
PROGRAM MAIN
VAR RETAIN
	rModuleOperaingSpeed		: REAL := 20;
END_VAR
VAR
	start:FB_CycleStart();	

	RelayOnTmr	: TOF;
	bSetRelay : BOOL;

	fbMeca500	: FB_MecaStateMachine;
	stModuleHmi : ST_ModuleHmi;
	stPlcCom	: ST_Module_PlcCom;
	stStation	: ST_Stations;
	fbLightTower : FB_ASMT60Functions;
	fbEventLogger	:FB_EventLogger;
	
	stCouplerData : ST_CouplerImagingData;
	stAssemblyData	: ST_Recipes;
	fbDataExchange		: FB_RecipeDataExchange;
	StAngleData : ST_AngleData; // RECEIVED ANGLE DATA FROM CPU 1
	fbGlueState	: FB_GlueState;


	fbDataExchangeRead	:FB_DataExchangeRead;
	bGroupRunStop AT %Q* : BOOL := TRUE;
	bSafetyError	 AT %I* : BOOL ;
	bErrorAck	AT %Q* : BOOL;
	SafetyAckOffTmr : TON;
	ErrorAckOffTmr	: TON;
	ResetButtonTmr1	: TON := (
		PT := T#1S);
	ResetButtonTmr2	: TON := (
		PT := T#0.5S);
	bSetOnce : BOOL := TRUE;
	bRinglightsSet	: BOOL;
	bAllowPowerOff	: BOOL;
	bLocksEngaged : BOOL;
	iProductionMainStep : INT;
	bAllowStationPrductionStart1To5 : BOOL;
	bAllowStationPrductionStart6To10 : BOOL;
	bLockAll		: BOOL;
	bUnlockGlueDoor : BOOL;
	LockTmr			: TON;
	sErrorText	: STRING;
	iRobotError	: INT;
	iCheckOperationality : INT;	
	iCheckStep	: INT;	
	bPlacingDone : BOOL;
	bAssemblyDone : BOOL;
	bCheckPassed : BOOL;
	iStepPosSave	: INT;
	bSet : BOOL;
	bNeedleSucceeded : BOOL;
END_VAR

start();


P_Heaters();

fbMeca500(stModuleHmi := stModuleHmi, stStations := stStation, stPlcCom := stPlcCom, stAssemblyData := stAssemblyData, bLocksEngaged := bLocksEngaged, stCouplerData := stCouplerData, rOperatingSpeed := rModuleOperaingSpeed, bNeedleSucceeded := bNeedleSucceeded);
fbDataExchange(sendRecipeData := stAssemblyData, stModuleHmi := stModuleHmi);
fbDataExchangeRead(stModuleHmi := stModuleHmi, stLaserPositionData => StAngleData);
ErrAck();
ResetLight();
HatchLight();
HatchLocks();
PowerBtn();
fbLightTower();
StartupTrig();
LaserPointers();
fbEventLogger(stModuleHmi:=stModuleHmi);
fbGlueState(stModuleHmi := stModuleHmi, stPlcCom := stPlcCom, bDetectionSucceeded := bNeedleSucceeded);


CASE iProductionMainStep OF
	0: IF stModuleHmi.bStartDetection THEN // LISÄÄ ROBOTIN ANTURIN TESTI
			fbMeca500.bExecuteNeedleTest := TRUE;
			stModuleHmi.bStartDetection := FALSE;
		END_IF
		
		IF stModuleHmi.bDispensingStageDone THEN
			iProductionMainStep := 1;
		ELSIF fbMeca500.bNeedleFailed THEN
			fbEventLogger.sErrorCode:='211';
			fbEventLogger.bRaiseAlarm[17]:= TRUE;
			stModuleHmi.bModuleProductionStart := FALSE;
			stModuleHmi.bProductionStart1To5 := FALSE;
			stModuleHmi.bProductionStart6To10 := FALSE;
			stModuleHmi.bProductionStageCompleted := FALSE;
			stModuleHmi.bProductionStartFailure := TRUE;
			iProductionMainStep := 0;
		END_IF

	1: IF stModuleHmi.bModuleProductionStart AND stPlcCom.stPlcComIn.bSafetyOk AND stPlcCom.stPlcComIn.bEstopOk AND stModuleHmi.bModuleStartupDone AND NOT stModuleHmi.bModuleFault THEN
			bLockAll := TRUE;
			stModuleHmi.bModulePlayPause := TRUE;
			stModuleHmi.bProductionStartFailure := FALSE;
			bUnlockGlueDoor := FALSE;
			ForceHoldersRelease();
			IF bLocksEngaged THEN
				iProductionMainStep := 2;
			ELSE
				iProductionMainStep := 30;
			END_IF
		END_IF 
	2: Trig.bOutfeedCam := TRUE;
		OutfeedLight(IN := TRUE);
		IF MAIN_VISION.fbOutfeedCam.bImagingDone THEN
			iProductionMainStep := 3;
			Trig.bOutfeedCam := FALSE;
			OutfeedLight(IN := FALSE);
		ELSIF MAIN_VISION.fbOutfeedCam.bError THEN
			iProductionMainStep := 30;
		END_IF
	3: IF NOT MAIN_VISION.fbOutfeedCam.bPalletRow1NotClear AND NOT MAIN_VISION.fbOutfeedCam.bPalletRow1NotClear THEN
			iProductionMainStep := 4;
			 Trig.bRejectCam := TRUE;
		ELSE
			iProductionMainStep := 30;
		END_IF
	4:	Trig.bRejectCam := TRUE;
		RejectLight(IN := TRUE);
		IF MAIN_VISION.fbRejectCam.bImagingDone THEN
			RejectLight(IN := FALSE);
			iProductionMainStep := 5;
			Trig.bRejectCam := FALSE;
		ELSIF MAIN_VISION.fbRejectCam.bError THEN
			iProductionMainStep := 30;
		END_IF
	5: IF NOT MAIN_VISION.fbRejectCam.bPalletRow1NotClear AND NOT MAIN_VISION.fbRejectCam.bPalletRow1NotClear THEN
			iProductionMainStep := 6;
		ELSE
			iProductionMainStep := 30;
		END_IF
	6: fbMeca500.bExecuteNeedleReTest := TRUE;
		iProductionMainStep := 7;
	7: ResetStns(All := TRUE, Stns1To5 := FALSE, Stns6To10 := FALSE);
		iProductionMainStep := 8;
		
	8: IF fbMeca500.bNeedleRecheckSucceeded (*AND MAIN_VISION.stPalletPosData.bMirrorPalletImagingSucceeded*)  THEN
			fbMeca500.bAllowStart := TRUE;
			IF stModuleHmi.bProductionStart1To5 AND stModuleHmi.bProductionStart6To10 THEN
				bAllowStationPrductionStart1To5 := TRUE;
				bAllowStationPrductionStart6To10 := TRUE;
				fbMeca500.bNewPlacingActive := TRUE;
				iProductionMainStep := 10;
			ELSIF stModuleHmi.bProductionStart1To5 THEN
				bAllowStationPrductionStart1To5 := TRUE;
				bAllowStationPrductionStart6To10 := FALSE; 
				fbMeca500.bNewPlacingActive := TRUE;
				iProductionMainStep := 20;
			END_IF
		ELSIF fbMeca500.bNeedleFailed THEN
			fbEventLogger.sErrorCode:='211';
			fbEventLogger.bRaiseAlarm[17]:= TRUE;
			stModuleHmi.bModuleProductionStart := FALSE;
			fbMeca500.bExecuteNeedleReTest := FALSE;
			stModuleHmi.bProductionStart1To5 := FALSE;
			stModuleHmi.bProductionStart6To10 := FALSE;
			stModuleHmi.bProductionStageCompleted := FALSE;
			stModuleHmi.bProductionStartFailure := TRUE;
			iProductionMainStep := 0;
		END_IF
		
	10: CheckAllPlacingState();
		IF bPlacingDone THEN
			stModuleHmi.bProductionStageCompleted := TRUE; // ALLOWS PAUSE BUTTON PRESS TO OPEN GLUING DOOR
			bPlacingDone := FALSE;
			fbMeca500.bNewPlacingActive := FALSE;
			iCheckStep := 0;
			iProductionMainStep := 11;
		END_IF
		
	11: IF fbMeca500.bDismountingActive THEN
			stModuleHmi.bProductionStageCompleted := FALSE;
		END_IF
		CheckAllAssemblyState();
		IF bAssemblyDone THEN
			bAssemblyDone := FALSE;
			stModuleHmi.bProductionStart1To5 := FALSE;
			stModuleHmi.bProductionStart6To10 := FALSE;
			bAllowStationPrductionStart1To5 := FALSE; 
			bAllowStationPrductionStart6To10 := FALSE; 
			stModuleHmi.bModuleProductionStart := FALSE;
			stModuleHmi.bProductionStageCompleted := FALSE;
			iProductionMainStep := 0;
			iCheckStep := 0;
		END_IF
		
	20: Check1To5PlacingState();
		IF bPlacingDone THEN
			stModuleHmi.bProductionStageCompleted := TRUE; // ALLOWS PAUSE BUTTON PRESS TO OPEN GLUING DOOR
			bPlacingDone := FALSE;
			iCheckStep := 0;
			iProductionMainStep := 21;
		END_IF
		
	21: IF fbMeca500.bDismountingActive THEN
			stModuleHmi.bProductionStageCompleted := FALSE;
		ELSIF stModuleHmi.bProductionStart6To10 THEN
			iStepPosSave := 22;
			iProductionMainStep := 60;
		END_IF
		Check1To5AssemblyState();
		IF bAssemblyDone THEN
			bAssemblyDone := FALSE;
			stModuleHmi.bProductionStart1To5 := FALSE;
			stModuleHmi.bProductionStart6To10 := FALSE;
			bAllowStationPrductionStart1To5 := FALSE; 
			bAllowStationPrductionStart6To10 := FALSE; 
			stModuleHmi.bModuleProductionStart := FALSE;
			stModuleHmi.bProductionStageCompleted := FALSE;
			iProductionMainStep := 0;
			iCheckStep := 0;
		END_IF
	22:	stModuleHmi.bProductionStageCompleted := FALSE;
		bAllowStationPrductionStart6To10 := TRUE;
		fbMeca500.bNewPlacingActive := TRUE;
		iProductionMainStep := 23;
		
	23: Check6To10PlacingState();
		IF bPlacingDone THEN
			fbMeca500.bNewPlacingActive := FALSE;
			stModuleHmi.bProductionStageCompleted := TRUE; // ALLOWS PAUSE BUTTON PRESS TO OPEN GLUING DOOR
			bPlacingDone := FALSE;
			iCheckStep := 0;
			iProductionMainStep := 24;
		END_IF
		
	24: Check1To5AssemblyState();
		IF bAssemblyDone THEN
			bAssemblyDone := FALSE;
			iCheckStep := 0;
			ResetStations();
			bAllowStationPrductionStart1To5 := FALSE; 
			stModuleHmi.bProductionStart1To5 := FALSE;
			iProductionMainStep := 25;
		END_IF
		
	25: IF fbMeca500.bDismountingActive THEN
			stModuleHmi.bProductionStageCompleted := FALSE;
		ELSIF stModuleHmi.bProductionStart1To5 THEN
			iStepPosSave := 26;
			iProductionMainStep := 50;
		END_IF
		Check6To10AssemblyState();
		IF bAssemblyDone THEN
			bAssemblyDone := FALSE;
			stModuleHmi.bProductionStart1To5 := FALSE;
			bAllowStationPrductionStart1To5 := FALSE; 
			bAllowStationPrductionStart6To10 := FALSE; 
			stModuleHmi.bModuleProductionStart := FALSE;
			stModuleHmi.bProductionStart6To10 := FALSE;
			ResetStations();
			stModuleHmi.bProductionStageCompleted := FALSE;
			iProductionMainStep := 0;
			iCheckStep := 0;
		END_IF
	26: fbMeca500.bNewPlacingActive := TRUE;
		bAllowStationPrductionStart1To5 := TRUE; 
		stModuleHmi.bProductionStageCompleted := FALSE;
		iProductionMainStep := 27;
		
	27: Check1To5PlacingState();
		IF bPlacingDone THEN
			fbMeca500.bNewPlacingActive := FALSE;
			stModuleHmi.bProductionStageCompleted := TRUE; // ALLOWS PAUSE BUTTON PRESS TO OPEN GLUING DOOR
			bPlacingDone := FALSE;
			iCheckStep := 0;
			iProductionMainStep := 28;
		END_IF
		
	28: Check6To10AssemblyState();
		IF bAssemblyDone THEN
			bAssemblyDone := FALSE;
			iCheckStep := 0;
			ResetStations();
			bAllowStationPrductionStart6To10 := FALSE; 
			stModuleHmi.bProductionStart6To10 := FALSE;
			iProductionMainStep := 21;
		END_IF
		
	30: bAssemblyDone := FALSE;
		OutfeedLight(IN := FALSE);
		RejectLight(IN := FALSE); 
		stModuleHmi.bProductionStartFailure := TRUE;
		fbMeca500.bExecuteNeedleTest := FALSE;
		stModuleHmi.bProductionStart1To5 := FALSE;
		stModuleHmi.bProductionStart6To10 := FALSE;
		bAllowStationPrductionStart1To5 := FALSE; 
		bAllowStationPrductionStart6To10 := FALSE; 
		stModuleHmi.bModuleProductionStart := FALSE;
		stModuleHmi.bProductionStageCompleted := FALSE;
		stModuleHmi.bModuleProductionStop := FALSE;
		iProductionMainStep := 0;
		iCheckStep := 0;
		
	50: Trig.bOutfeedCam := TRUE;				// Check for pallet positions 1 to 5
		OutfeedLight(IN := TRUE);
		ResetStns(All := FALSE, Stns1To5 := FALSE, Stns6To10 := TRUE);
		IF MAIN_VISION.fbOutfeedCam.bImagingDone THEN
			OutfeedLight(IN := FALSE);
			iProductionMainStep := 51;
			Trig.bOutfeedCam := FALSE;
		ELSIF MAIN_VISION.fbOutfeedCam.bError THEN
			iProductionMainStep := 58;
		END_IF
		
	51: IF NOT MAIN_VISION.fbOutfeedCam.bPalletRow1NotClear THEN // LISÄÄ 		
			Trig.bRejectCam := TRUE;	
			RejectLight(IN := TRUE);
			iProductionMainStep := 52;
		ELSE
			iProductionMainStep := 58;
		END_IF
	52:IF MAIN_VISION.fbRejectCam.bImagingDone THEN
			iProductionMainStep := 53;
			RejectLight(IN := FALSE);
			Trig.bRejectCam := FALSE;
		ELSIF MAIN_VISION.fbRejectCam.bError THEN
			iProductionMainStep := 58;
		END_IF
	53: IF NOT MAIN_VISION.fbRejectCam.bPalletRow1NotClear THEN // LISÄÄ 		
			fbMeca500.bExecuteNeedleTest := TRUE;	
			iProductionMainStep := 54;
		ELSE
			iProductionMainStep := 58;
		END_IF
	
	54: IF bNeedleSucceeded (*AND MAIN_VISION.stPalletPosData.bMirrorPalletImagingSucceeded *)THEN
			iProductionMainStep := iStepPosSave;
		ELSIF fbMeca500.bNeedleFailed THEN
			iProductionMainStep := 58;
		END_IF
		
	58: iProductionMainStep := iStepPosSave-1;
		bAllowStationPrductionStart1To5 := FALSE; 
		OutfeedLight(IN := FALSE);
		RejectLight(IN := FALSE);
		stModuleHmi.bProductionStart1To5 := FALSE;
		Err.Err; //404
		
	60: Trig.bOutfeedCam := TRUE;				// Check for pallet positions 6 to 10
		ResetStns(All := FALSE, Stns1To5 := FALSE, Stns6To10 := TRUE);
		OutfeedLight(IN := TRUE);
		IF MAIN_VISION.fbOutfeedCam.bImagingDone THEN
			OutfeedLight(IN := FALSE);
			iProductionMainStep := 61;
			Trig.bOutfeedCam := FALSE;
		ELSIF MAIN_VISION.fbOutfeedCam.bError THEN
			iProductionMainStep := 68;
		END_IF
		
	61: IF NOT MAIN_VISION.fbOutfeedCam.bPalletRow2NotClear THEN // LISÄÄ fbMeca500.bExecuteNeedleTest := TRUE;	
			Trig.bRejectCam := TRUE;
			RejectLight(IN := TRUE);
			iProductionMainStep := 62;
		ELSE
			iProductionMainStep := 68;
		END_IF
	62: IF MAIN_VISION.fbRejectCam.bImagingDone THEN
			iProductionMainStep := 63;
			RejectLight(IN := FALSE);
			Trig.bRejectCam := FALSE;
		ELSIF MAIN_VISION.fbRejectCam.bError THEN
			iProductionMainStep := 68;
		END_IF
	63: IF NOT MAIN_VISION.fbRejectCam.bPalletRow2NotClear THEN // LISÄÄ 		
			fbMeca500.bExecuteNeedleTest := TRUE;	
			iProductionMainStep := 64;
		ELSE
			iProductionMainStep := 68;
		END_IF
	64: IF bNeedleSucceeded (*AND MAIN_VISION.stPalletPosData.bMirrorPalletImagingSucceeded *)THEN
			iProductionMainStep := iStepPosSave;
		ELSIF fbMeca500.bNeedleFailed THEN
			iProductionMainStep := 68;
		END_IF
		
	68:	iProductionMainStep := iStepPosSave-1;
		OutfeedLight(IN := FALSE);
		RejectLight(IN := FALSE);
		bAllowStationPrductionStart6To10 := FALSE; 
		stModuleHmi.bProductionStart6To10 := FALSE;
		Err.Err; // 404
		
END_CASE

IF stModuleHmi.bModuleProductionStop THEN
	iProductionMainStep := 30;
END_IF




////STATIONS
stStation.fbSts1(iStationId := 1, 
	stMirrorData := MAIN_VISION.stMirrorDataSts1, 
	stLaserData := StAngleData.stLaserData1,
	stModuleHmi := stModuleHmi, 
	stModulePlcCom := stPlcCom,
	bActivateStation := stModuleHmi.Stations.bActivateStation1,
	bAllowStart := bAllowStationPrductionStart1To5,
	bReleaseHolders := stModuleHmi.Stations.bReleaseHolders1,
	sTimeLeft => stModuleHmi.Stations.tAssemmblyTime1,
	bTrigAngCam => stAssemblyData.Station1To5.bTrigCam1);

stStation.fbSts2(iStationId := 2, 
	stMirrorData := MAIN_VISION.stMirrorDatasts2, 
	stLaserData := StAngleData.stLaserData2,
	stModuleHmi := stModuleHmi, 
	stModulePlcCom := stPlcCom,
	bAllowStart := bAllowStationPrductionStart1To5,
	bActivateStation := stModuleHmi.Stations.bActivateStation2,
	bReleaseHolders := stModuleHmi.Stations.bReleaseHolders2,
	sTimeLeft => stModuleHmi.Stations.tAssemmblyTime2,
	bTrigAngCam => stAssemblyData.Station1To5.bTrigCam2);
	
stStation.fbSts3(iStationId := 3, 
	stMirrorData := MAIN_VISION.stMirrorDatasts3, 
	stLaserData := StAngleData.stLaserData3,
	stModuleHmi := stModuleHmi, 
	stModulePlcCom := stPlcCom,
	bAllowStart := bAllowStationPrductionStart1To5,
	bActivateStation := stModuleHmi.Stations.bActivateStation3,
	bReleaseHolders := stModuleHmi.Stations.bReleaseHolders3,
	sTimeLeft => stModuleHmi.Stations.tAssemmblyTime3,
	bTrigAngCam => stAssemblyData.Station1To5.bTrigCam3);

stStation.fbSts4(iStationId := 4, 
	stMirrorData := MAIN_VISION.stMirrorDatasts4, 
	stLaserData := StAngleData.stLaserData4,
	stModuleHmi := stModuleHmi, 
	stModulePlcCom := stPlcCom,
	bAllowStart := bAllowStationPrductionStart1To5,
	bActivateStation := stModuleHmi.Stations.bActivateStation4,
	bReleaseHolders := stModuleHmi.Stations.bReleaseHolders4,
	sTimeLeft => stModuleHmi.Stations.tAssemmblyTime4,
	bTrigAngCam => stAssemblyData.Station1To5.bTrigCam4);
	
stStation.fbSts5(iStationId := 5, 
	stMirrorData := MAIN_VISION.stMirrorDatasts5, 
	stLaserData := StAngleData.stLaserData5,
	stModuleHmi := stModuleHmi, 
	stModulePlcCom := stPlcCom,
	bAllowStart := bAllowStationPrductionStart1To5,
	bActivateStation := stModuleHmi.Stations.bActivateStation5,
	bReleaseHolders := stModuleHmi.Stations.bReleaseHolders5,
	sTimeLeft => stModuleHmi.Stations.tAssemmblyTime5,
	bTrigAngCam => stAssemblyData.Station1To5.bTrigCam5);
	
stStation.fbSts6(iStationId := 6, 
	stMirrorData := MAIN_VISION.stMirrorDatasts6, 
	stLaserData := StAngleData.stLaserData6,
	stModuleHmi := stModuleHmi, 
	stModulePlcCom := stPlcCom,
	bAllowStart := bAllowStationPrductionStart6To10,
	bActivateStation := stModuleHmi.Stations.bActivateStation6,
	bReleaseHolders := stModuleHmi.Stations.bReleaseHolders6,
	sTimeLeft => stModuleHmi.Stations.tAssemmblyTime6,
	bTrigAngCam => stAssemblyData.Station5To10.bTrigCam6);
	
stStation.fbSts7(iStationId := 7, 
	stMirrorData := MAIN_VISION.stMirrorDatasts7, 
	stLaserData := StAngleData.stLaserData7,
	stModuleHmi := stModuleHmi, 
	stModulePlcCom := stPlcCom,
	bAllowStart := bAllowStationPrductionStart6To10,
	bActivateStation := stModuleHmi.Stations.bActivateStation7,
	bReleaseHolders := stModuleHmi.Stations.bReleaseHolders7,
	sTimeLeft => stModuleHmi.Stations.tAssemmblyTime7,
	bTrigAngCam => stAssemblyData.Station5To10.bTrigCam7);
	
stStation.fbSts8(iStationId := 8, 
	stMirrorData := MAIN_VISION.stMirrorDatasts8, 
	stLaserData := StAngleData.stLaserData8,
	stModuleHmi := stModuleHmi, 
	stModulePlcCom := stPlcCom,
	bAllowStart := bAllowStationPrductionStart6To10,
	bActivateStation := stModuleHmi.Stations.bActivateStation8,
	bReleaseHolders := stModuleHmi.Stations.bReleaseHolders8,
	sTimeLeft => stModuleHmi.Stations.tAssemmblyTime8,
	bTrigAngCam => stAssemblyData.Station5To10.bTrigCam8);
	
stStation.fbSts9(iStationId := 9, 
	stMirrorData := MAIN_VISION.stMirrorDatasts9, 
	stLaserData := StAngleData.stLaserData9,
	stModuleHmi := stModuleHmi, 
	stModulePlcCom := stPlcCom,
	bAllowStart := bAllowStationPrductionStart6To10,
	bActivateStation := stModuleHmi.Stations.bActivateStation9,
	bReleaseHolders := stModuleHmi.Stations.bReleaseHolders9,
	sTimeLeft => stModuleHmi.Stations.tAssemmblyTime9,
	bTrigAngCam => stAssemblyData.Station5To10.bTrigCam9);
	
stStation.fbSts10(iStationId := 10, 
	stMirrorData := MAIN_VISION.stMirrorDatasts10, 
	stLaserData := StAngleData.stLaserData10,
	stModuleHmi := stModuleHmi, 
	stModulePlcCom := stPlcCom,
	bAllowStart := bAllowStationPrductionStart6To10,
	bActivateStation := stModuleHmi.Stations.bActivateStation10,
	bReleaseHolders := stModuleHmi.Stations.bReleaseHolders10,
	sTimeLeft => stModuleHmi.Stations.tAssemmblyTime10,
	bTrigAngCam => stAssemblyData.Station5To10.bTrigCam10);

ACTION Check1To5AssemblyState:

	CASE iCheckStep OF
		0: iCheckStep := 1;

		1:	IF stModuleHmi.Stations.bActivateStation1 THEN
					iCheckStep := 2;
			END_IF
		2:	IF stModuleHmi.Stations.bActivateStation2 THEN
				iCheckStep := 3;
			END_IF
		3:	IF stModuleHmi.Stations.bActivateStation3 THEN
					iCheckStep := 4;
			END_IF
		4:	IF stModuleHmi.Stations.bActivateStation4 THEN
					iCheckStep := 5;
			END_IF
		5:	IF stModuleHmi.Stations.bActivateStation5 THEN
					iCheckStep := 11;
			END_IF
			
		6:	IF stModuleHmi.Stations.bActivateStation6 THEN
					iCheckStep := 7;
			END_IF
		7:	IF stModuleHmi.Stations.bActivateStation7 THEN
					iCheckStep := 8;
			END_IF
		8:	IF stModuleHmi.Stations.bActivateStation8 THEN
					iCheckStep := 9;
			END_IF
		9:	IF stModuleHmi.Stations.bActivateStation9 THEN
					iCheckStep := 10;
			END_IF
		10: IF stModuleHmi.Stations.bActivateStation10 THEN
					iCheckStep := 11;
			END_IF
		11: bAssemblyDone := TRUE;
			iCheckStep := 0;
			
	END_CASE
END_ACTION

ACTION Check1To5PlacingState:


	CASE iCheckStep OF
		0:	iCheckStep := 1;
		1:	IF stModuleHmi.Stations.bActivateStation1 THEN
				IF stStation.fbSts1.bPlacingDone THEN
					iCheckStep := 2;
				END_IF
			ELSE
					iCheckStep := 2;
			END_IF
		2:	IF stModuleHmi.Stations.bActivateStation2 THEN
				IF stStation.fbSts2.bPlacingDone THEN
					iCheckStep := 3;
				END_IF
			ELSE
					iCheckStep := 3;
			END_IF
		3:	IF stModuleHmi.Stations.bActivateStation3 THEN
				IF stStation.fbSts3.bPlacingDone THEN
					iCheckStep := 4;
				END_IF
			ELSE
					iCheckStep := 4;
			END_IF
		4:	IF stModuleHmi.Stations.bActivateStation4 THEN
				IF stStation.fbSts4.bPlacingDone THEN
					iCheckStep := 5;
				END_IF
			ELSE
					iCheckStep := 5;
			END_IF
			
		5:	IF stModuleHmi.Stations.bActivateStation5 THEN
				IF stStation.fbSts5.bPlacingDone THEN
					iCheckStep := 11;
				END_IF
			ELSE
					iCheckStep := 11;
			END_IF
			
		6:	IF stModuleHmi.Stations.bActivateStation6 THEN
				IF stStation.fbSts6.bPlacingDone THEN
					iCheckStep := 7;
				END_IF
			ELSE
					iCheckStep := 7;
			END_IF
		7:	IF stModuleHmi.Stations.bActivateStation7 THEN
				IF stStation.fbSts7.bPlacingDone THEN
					iCheckStep := 8;
				END_IF
			ELSE
					iCheckStep := 8;
			END_IF
		8:	IF stModuleHmi.Stations.bActivateStation8 THEN
				IF stStation.fbSts8.bPlacingDone THEN
					iCheckStep := 9;
				END_IF
			ELSE
					iCheckStep := 9;
			END_IF
		9:	IF stModuleHmi.Stations.bActivateStation9 THEN
				IF stStation.fbSts9.bPlacingDone THEN
					iCheckStep := 10;
				END_IF
			ELSE
					iCheckStep := 10;
			END_IF
		10: IF stModuleHmi.Stations.bActivateStation10 THEN
				IF stStation.fbSts10.bPlacingDone THEN
					iCheckStep := 11;
				END_IF
			ELSE
					iCheckStep := 11;
			END_IF
		11: bPlacingDone := TRUE;
			iCheckStep := 0;
			
	END_CASE
END_ACTION

ACTION Check6To10AssemblyState:

	CASE iCheckStep OF
		0: iCheckStep := 6;

		1:	IF stModuleHmi.Stations.bActivateStation1 THEN
					iCheckStep := 2;
			END_IF
		2:	IF stModuleHmi.Stations.bActivateStation2 THEN
				iCheckStep := 3;
			END_IF
		3:	IF stModuleHmi.Stations.bActivateStation3 THEN
					iCheckStep := 4;
			END_IF
		4:	IF stModuleHmi.Stations.bActivateStation4 THEN
					iCheckStep := 5;
			END_IF
		5:	IF stModuleHmi.Stations.bActivateStation5 THEN
					iCheckStep := 11;
			END_IF
			
		6:	IF stModuleHmi.Stations.bActivateStation6 THEN
					iCheckStep := 7;
			END_IF
		7:	IF stModuleHmi.Stations.bActivateStation7 THEN
					iCheckStep := 8;
			END_IF
		8:	IF stModuleHmi.Stations.bActivateStation8 THEN
					iCheckStep := 9;
			END_IF
		9:	IF stModuleHmi.Stations.bActivateStation9 THEN
					iCheckStep := 10;
			END_IF
		10: IF stModuleHmi.Stations.bActivateStation10 THEN
					iCheckStep := 11;
			END_IF
		11: bAssemblyDone := TRUE;
			iCheckStep := 0;
			
	END_CASE
END_ACTION

ACTION Check6To10PlacingState:


	CASE iCheckStep OF
		0:	iCheckStep := 6;
		1:	IF stModuleHmi.Stations.bActivateStation1 THEN
				IF stStation.fbSts1.bPlacingDone THEN
					iCheckStep := 2;
				END_IF
			ELSE
					iCheckStep := 2;
			END_IF
		2:	IF stModuleHmi.Stations.bActivateStation2 THEN
				IF stStation.fbSts2.bPlacingDone THEN
					iCheckStep := 3;
				END_IF
			ELSE
					iCheckStep := 3;
			END_IF
		3:	IF stModuleHmi.Stations.bActivateStation3 THEN
				IF stStation.fbSts3.bPlacingDone THEN
					iCheckStep := 4;
				END_IF
			ELSE
					iCheckStep := 4;
			END_IF
		4:	IF stModuleHmi.Stations.bActivateStation4 THEN
				IF stStation.fbSts4.bPlacingDone THEN
					iCheckStep := 5;
				END_IF
			ELSE
					iCheckStep := 5;
			END_IF
			
		5:	IF stModuleHmi.Stations.bActivateStation5 THEN
				IF stStation.fbSts5.bPlacingDone THEN
					iCheckStep := 11;
				END_IF
			ELSE
					iCheckStep := 11;
			END_IF
			
		6:	IF stModuleHmi.Stations.bActivateStation6 THEN
				IF stStation.fbSts6.bPlacingDone THEN
					iCheckStep := 7;
				END_IF
			ELSE
					iCheckStep := 7;
			END_IF
		7:	IF stModuleHmi.Stations.bActivateStation7 THEN
				IF stStation.fbSts7.bPlacingDone THEN
					iCheckStep := 8;
				END_IF
			ELSE
					iCheckStep := 8;
			END_IF
		8:	IF stModuleHmi.Stations.bActivateStation8 THEN
				IF stStation.fbSts8.bPlacingDone THEN
					iCheckStep := 9;
				END_IF
			ELSE
					iCheckStep := 9;
			END_IF
		9:	IF stModuleHmi.Stations.bActivateStation9 THEN
				IF stStation.fbSts9.bPlacingDone THEN
					iCheckStep := 10;
				END_IF
			ELSE
					iCheckStep := 10;
			END_IF
		10: IF stModuleHmi.Stations.bActivateStation10 THEN
				IF stStation.fbSts10.bPlacingDone THEN
					iCheckStep := 11;
				END_IF
			ELSE
					iCheckStep := 11;
			END_IF
		11: bPlacingDone := TRUE;
			iCheckStep := 0;
			
	END_CASE
END_ACTION

ACTION CheckAllAssemblyState:

	CASE iCheckStep OF
		0: iCheckStep := 1;

		1:	IF stModuleHmi.Stations.bActivateStation1 THEN
					iCheckStep := 2;
			END_IF
		2:	IF stModuleHmi.Stations.bActivateStation2 THEN
				iCheckStep := 3;
			END_IF
		3:	IF stModuleHmi.Stations.bActivateStation3 THEN
					iCheckStep := 4;
			END_IF
		4:	IF stModuleHmi.Stations.bActivateStation4 THEN
					iCheckStep := 5;
			END_IF
		5:	IF stModuleHmi.Stations.bActivateStation5 THEN
					iCheckStep := 6;
			END_IF
			
		6:	IF stModuleHmi.Stations.bActivateStation6 THEN
					iCheckStep := 7;
			END_IF
		7:	IF stModuleHmi.Stations.bActivateStation7 THEN
					iCheckStep := 8;
			END_IF
		8:	IF stModuleHmi.Stations.bActivateStation8 THEN
					iCheckStep := 9;
			END_IF
		9:	IF stModuleHmi.Stations.bActivateStation9 THEN
					iCheckStep := 10;
			END_IF
		10: IF stModuleHmi.Stations.bActivateStation10 THEN
					iCheckStep := 11;
			END_IF
		11: bAssemblyDone := TRUE;
			iCheckStep := 0;
			
	END_CASE
END_ACTION

ACTION CheckAllPlacingState:


	CASE iCheckStep OF
		0:	iCheckStep := 1;
		1:	IF stModuleHmi.Stations.bActivateStation1 THEN
				IF stStation.fbSts1.bPlacingDone THEN
					iCheckStep := 2;
				END_IF
			ELSE
					iCheckStep := 2;
			END_IF
		2:	IF stModuleHmi.Stations.bActivateStation2 THEN
				IF stStation.fbSts2.bPlacingDone THEN
					iCheckStep := 3;
				END_IF
			ELSE
					iCheckStep := 3;
			END_IF
		3:	IF stModuleHmi.Stations.bActivateStation3 THEN
				IF stStation.fbSts3.bPlacingDone THEN
					iCheckStep := 4;
				END_IF
			ELSE
					iCheckStep := 4;
			END_IF
		4:	IF stModuleHmi.Stations.bActivateStation4 THEN
				IF stStation.fbSts4.bPlacingDone THEN
					iCheckStep := 5;
				END_IF
			ELSE
					iCheckStep := 5;
			END_IF
			
		5:	IF stModuleHmi.Stations.bActivateStation5 THEN
				IF stStation.fbSts5.bPlacingDone THEN
					iCheckStep := 6;
				END_IF
			ELSE
					iCheckStep := 6;
			END_IF
			
		6:	IF stModuleHmi.Stations.bActivateStation6 THEN
				IF stStation.fbSts6.bPlacingDone THEN
					iCheckStep := 7;
				END_IF
			ELSE
					iCheckStep := 7;
			END_IF
		7:	IF stModuleHmi.Stations.bActivateStation7 THEN
				IF stStation.fbSts7.bPlacingDone THEN
					iCheckStep := 8;
				END_IF
			ELSE
					iCheckStep := 8;
			END_IF
		8:	IF stModuleHmi.Stations.bActivateStation8 THEN
				IF stStation.fbSts8.bPlacingDone THEN
					iCheckStep := 9;
				END_IF
			ELSE
					iCheckStep := 9;
			END_IF
		9:	IF stModuleHmi.Stations.bActivateStation9 THEN
				IF stStation.fbSts9.bPlacingDone THEN
					iCheckStep := 10;
				END_IF
			ELSE
					iCheckStep := 10;
			END_IF
		10: IF stModuleHmi.Stations.bActivateStation10 THEN
				IF stStation.fbSts10.bPlacingDone THEN
					iCheckStep := 11;
				END_IF
			ELSE
					iCheckStep := 11;
			END_IF
		11: bPlacingDone := TRUE;
			
	END_CASE
END_ACTION

ACTION CheckCompatibility:

IF stModuleHmi.bProductionStart1To5 AND stModuleHmi.bProductionStart6To10 THEN
	IF stAssemblyData.Station1To5.rGalvoThickness = stAssemblyData.Station5To10.rGalvoThickness THEN
		bCheckPassed := TRUE;
	ELSE
		bCheckPassed := FALSE;
	END_IF
END_IF
END_ACTION

METHOD ErrAck : BOOL
VAR_INPUT
END_VAR
IF bSafetyError AND NOT bErrorAck OR SafetyAckOffTmr.Q THEN
	SafetyAckOffTmr.IN := FALSE;
	bErrorAck := TRUE;
	ErrorAckOffTmr.IN := TRUE;
ELSIF NOT bSafetyError THEN
	SafetyAckOffTmr.IN := FALSE;
END_IF

IF bErrorAck AND ErrorAckOffTmr.Q THEN
	ErrorAckOffTmr.IN := FALSE;
	bErrorAck := FALSE;
	SafetyAckOffTmr.IN := TRUE;
END_IF
SafetyAckOffTmr(PT := T#2S);
ErrorAckOffTmr(PT := T#0.5S);
END_METHOD

ACTION ErrorList:
CASE iRobotError OF
0:	  sErrorText := 'NO_ERROR';
1000: sErrorText := 'COMMAND_BUFFER_IS_FULL';
1001: sErrorText := 'UNKNOWN_COMMAND';
1002: sErrorText := 'SYNTAX_ERROR';
1003: sErrorText := 'ARGUMENT_ERROR';
1005: sErrorText := 'THE_ROBOT_IS_NOT_ACTIVATED';
1006: sErrorText := 'THE_ROBOT_IS_NOT_HOMED';
1007: sErrorText := 'JOINT_OVER_LIMIT';
1010: sErrorText := 'LINEAR_MOVE_BLOCKED_BY_ROTATION';
1011: sErrorText := 'THE_ROBOT_IS_IN_ERROR';
1012: sErrorText := 'SINGULARITY_DETECTED';
1013: sErrorText := 'ACTIVATION_FAILED';
1014: sErrorText := 'HOMING_FAILED';
1016: sErrorText := 'POSE_OUT_OF_REACH';
1022: sErrorText := 'PROGRAM_SAVING_FAILED_1';
1023: sErrorText := 'IGNORING_COMMAND_FOR_OFFLINE_MODE';
1024: sErrorText := 'MASTERING_NEEDED';
1025: sErrorText := 'RESET_ERROR_NOT_POSSIBLE';
1026: sErrorText := 'DeactivatedIVATION_NEEDED';
1027: sErrorText := 'CHANGE_SIMULATION_MODE_FAILED';
1030: sErrorText := 'ALREADY_SAVING';
1031: sErrorText := 'PROGRAM_SAVING_ABORTED';
1033: sErrorText := 'START_CONF_MISMATCH';
1038: sErrorText := 'ERR_NO_GRIPPER_CONNECTED';
1040: sErrorText := 'COMMAND_FAILED';
1041: sErrorText := 'NO_VBOX';
1042: sErrorText := 'EXT_TOOL_SIM_MUST_Deactivated';
1043: sErrorText := 'IO_BANK_NOT_PRESENT';
1044: sErrorText := 'VACUUM_MODULE_NOT_PRESENT';
3005: sErrorText := 'MOTION_ERROR';
3006: sErrorText := 'DRIVE_ERROR';
3009: sErrorText := 'INIT_FAILED';
3014: sErrorText := 'ERROR_SAVING';
3020: sErrorText := 'INVALID_OFFLINE_PROGRAM';
3025: sErrorText := 'GRIPPER_ERROR';
3026: sErrorText := 'MAINTENANCE_CHECK_DISCOVERY';
3029: sErrorText := 'EXCESSIVE_TORQUE';
3037: sErrorText := 'PNEUMATIC_ERROR';
3039: sErrorText := 'EXT_TOOL_NEED_UPDATE';
3041: sErrorText := 'IMMINENT_COLLISION';
3043: sErrorText := 'IO_PORT_PACKET_LOST';
3044: sErrorText := 'IO_PORT_COMM_ERROR';
3045: sErrorText := 'IMMINENT_COLLISION_DETECTED';
3046: sErrorText := 'POWERSUPPLY_ERROR';
3047: sErrorText := 'SAFE_MODE_BOOT';
3049: sErrorText := 'AT_WORKZONE_LIMIT';
END_CASE
END_ACTION

ACTION ForceHoldersRelease:

CASE iCheckOperationality OF
	0: iCheckOperationality := 1;
	1:	stStation.fbSts1.bReleaseHolders := TRUE;
		iCheckOperationality := 2;
	2: stStation.fbSts2.bReleaseHolders := TRUE;
		iCheckOperationality := 3; 
	3: stStation.fbSts3.bReleaseHolders := TRUE;
		iCheckOperationality := 4;
	4: stStation.fbSts4.bReleaseHolders := TRUE;
		iCheckOperationality := 5;
	5: stStation.fbSts5.bReleaseHolders := TRUE;
		iCheckOperationality := 6;
	6: stStation.fbSts6.bReleaseHolders := TRUE;
		iCheckOperationality := 7;
	7: stStation.fbSts7.bReleaseHolders := TRUE;
		iCheckOperationality := 8;
	8: stStation.fbSts8.bReleaseHolders := TRUE;
		iCheckOperationality := 9;
	9: stStation.fbSts9.bReleaseHolders := TRUE;
		iCheckOperationality := 10;
	10:stStation.fbSts10.bReleaseHolders := TRUE;
		iCheckOperationality := 0;
END_CASE
END_ACTION

METHOD GluingState
VAR_INPUT
END_VAR
END_METHOD

